   VAR 
      statConfiguration : "typeLPMLV30_Configuration" := ([12(false), 20(true)], [32(0)]);   // FB configuration
      statUnitModeChangeRequest : Bool := false;   // TRUE: Enable change into requested unit mode
      statCmdChangeRequest : Bool := false;   // TRUE: Enable change into requested state
      statFirstCycle { ExternalAccessible := 'False'; ExternalVisible := 'False'; ExternalWritable := 'False'} : Bool := true;   // First cycle of run
      statSCOld { ExternalAccessible := 'False'; ExternalVisible := 'False'; ExternalWritable := 'False'} : Bool := false;   // For edge detection
      statUnitMode { ExternalAccessible := 'False'; ExternalVisible := 'False'; ExternalWritable := 'False'} : DInt := "LPMLV30_MODE_MANUAL";   // Current command mode
      statUnitModeOld { ExternalAccessible := 'False'; ExternalVisible := 'False'; ExternalWritable := 'False'} : DInt := "LPMLV30_MODE_MANUAL";   // For edge detection
      statUnitModeCurrentInternal { ExternalAccessible := 'False'; ExternalVisible := 'False'; ExternalWritable := 'False'} : DInt := "LPMLV30_MODE_MANUAL";   // Current internal Mode
      statUnitModeCurrentInternalOld { ExternalAccessible := 'False'; ExternalVisible := 'False'; ExternalWritable := 'False'} : DInt := "LPMLV30_MODE_INVALID";   // For edge detection
      statStateCurrentOld { ExternalAccessible := 'False'; ExternalVisible := 'False'; ExternalWritable := 'False'} : DInt := "LPMLV30_STATE_STOPPED";   // For edge detection
      statStateInternal { ExternalAccessible := 'False'; ExternalVisible := 'False'; ExternalWritable := 'False'} : DInt := "LPMLV30_STATE_STOPPED";   // Current internal state
      statStateInternalOld { ExternalAccessible := 'False'; ExternalVisible := 'False'; ExternalWritable := 'False'} : DInt := "LPMLV30_STATE_UNDEFINED";   // For edge detection
      statCntrlCmdOld { ExternalAccessible := 'False'; ExternalVisible := 'False'; ExternalWritable := 'False'} : DInt := "LPMLV30_CMD_UNDEFINED";   // For edge detection
      statStatesInCurrentMode : Struct   // Copied from configuration
         clearing : Bool;
         stopped : Bool;
         starting : Bool;
         idle : Bool;
         suspended : Bool;
         execute : Bool;
         stopping : Bool;
         aborting : Bool;
         aborted : Bool;
         holding : Bool;
         held : Bool;
         unholding : Bool;
         suspending : Bool;
         unsuspending : Bool;
         resetting : Bool;
         completing : Bool;
         complete : Bool;
      END_STRUCT;
      statBooleanInterfaceModeOld { ExternalAccessible := 'False'; ExternalVisible := 'False'; ExternalWritable := 'False'} : DWord;   // For edge detection
      statBooleanInterfaceCmdOld { ExternalAccessible := 'False'; ExternalVisible := 'False'; ExternalWritable := 'False'} : Word;   // For edge detection
      statCmdChangeRequestOld : Bool := false;   // For edge detection
      statUnitModeChangeRequestOld : Bool := false;   // For edge detection
   END_VAR

   VAR_TEMP 
      tempCntrlCmd : DInt;   // Temporary control command
      tempBooleanInterfaceMode : DWord;   // Status of boolean Mode inputs if  boolean interface is active
      tempBooleanInterfaceCmd : Word;   // Status of boolean Cmd inputs except abort and stop if  boolean interface is active
      tempSCInternal : Bool;   // Internal state complete
      tempRetVal : Int;   // Tag for system function
      tempDiagnosticsBufferIndex : Int;   // Index of actual diagnostics buffer entry
      tempDiagnosticsBufferIndexSC : Int;   // Index of actual diagnostics buffer entry for SC messages
      tempDiagnosticsBufferIndexCmd : Int;   // Index of actual diagnostics buffer entry for control command messages
   END_VAR

   VAR CONSTANT 
      MSG_NO_MESSAGE : Byte := 16#00;   // Initial value
      MSG_MODE_CHANGED_SUCCESSFULLY : Byte := 16#01;   // Unit mode changed successfully
      MSG_STATE_CHANGED_SUCCESSFULLY : Byte := 16#02;   // State changed successfully
      MSG_MODE_ALREADY_ACTIVE : Byte := 16#03;   // Requested unit mode already active
      MSG_MODE_NOT_DEFINED : Byte := 16#80;   // Unit mode not defined
      MSG_CMD_NOT_DEFINED : Byte := 16#81;   // Control command not defined
      MSG_REQ_MODE_NOT_CONFIGURED : Byte := 16#82;   // Requested unit mode not configured
      MSG_MODE_TRANSITION_NOT_ALLOWED : Byte := 16#83;   // Unit mode transition not allowed
      MSG_CMD_NOT_ALLOWED : Byte := 16#84;   // Control command in this state not allowed
      MSG_SC_NOT_ALLOWED : Byte := 16#85;   // SC in this state not allowed
      MSG_STATE_CONFIG_FORCED : Byte := 16#86;   // State configuration forced to OMAC standard (corrected configuration -> FB output StatesDisabled)
   END_VAR


BEGIN
	//============================================================================================================
	// SIEMENS AG
	// (c)Copyright 2015 All Rights Reserved
	//------------------------------------------------------------------------------------------------------------
	// Library: LPMLV30
	// Tested with: S7-1200 with FW version V4.1, S7-1500 with FW version V1.7
	// Engineering: TIA Portal V13 SP1
	// Restrictions: ---
	// Requirements: S7-1200 / S7-1500
	// Functionality: Management of unit modes and states according to ISA TR88.00.02 - June 4, 2014
	//------------------------------------------------------------------------------------------------------------
	// Change log table:
	// Version  Date        Expert in charge    Changes applied
	// 03.00.01 29.05.2015  RK                  First released version 
	//============================================================================================================
	// Function block: LPMLV30_UnitModeStateManager
	//============================================================================================================
	
	IF NOT #statCmdChangeRequest AND #statCmdChangeRequestOld THEN // Falling edge CmdChangeRequest
	  #statCntrlCmdOld := "LPMLV30_CMD_UNDEFINED";
	END_IF;
	#statCmdChangeRequestOld := #statCmdChangeRequest;
	
	IF NOT #statUnitModeChangeRequest AND #statUnitModeChangeRequestOld THEN // Falling edge UnitModeChangeRequest
	  #statUnitModeOld := "LPMLV30_MODE_INVALID";
	END_IF;
	#statUnitModeChangeRequestOld := #statUnitModeChangeRequest;
	
	#tempDiagnosticsBufferIndex    := #diagnostics.bufferIndex; // Work with temporary variable during block execution
	#tempDiagnosticsBufferIndexSC  := -1;
	#tempDiagnosticsBufferIndexCmd := -1;
	
	IF #statFirstCycle THEN // Initialize values in first cycle
	  #tempDiagnosticsBufferIndex := -1;
	
	  #statConfiguration := #configuration; // Copy configuration from input
	  #statConfiguration.disabledUnitModes["LPMLV30_MODE_MANUAL"] := FALSE; // Unit mode Manual is mandatory
	  
	  // Initialize unit mode
	  #statUnitMode                   := "LPMLV30_MODE_MANUAL";
	  #statUnitModeOld                := "LPMLV30_MODE_MANUAL";
	  #UnitModeCurrent                := "LPMLV30_MODE_MANUAL";
	  #statUnitModeCurrentInternal    := "LPMLV30_MODE_MANUAL";
	  #statUnitModeCurrentInternalOld := "LPMLV30_MODE_INVALID";
	  #statBooleanInterfaceModeOld    := 0;
	  
	  // Initialize state
	  #StateCurrent         := "LPMLV30_STATE_STOPPED";
	  #StateRequested       := "LPMLV30_STATE_STOPPED";
	  #statStateInternal    := "LPMLV30_STATE_STOPPED";
	  #statStateInternalOld := "LPMLV30_STATE_UNDEFINED";
	  #statStateCurrentOld  := "LPMLV30_STATE_STOPPED";
	  
	  // Initialize control command
	  #tempCntrlCmd               := "LPMLV30_CMD_UNDEFINED";
	  #statCntrlCmdOld            := "LPMLV30_CMD_UNDEFINED";
	  #statBooleanInterfaceCmdOld := 0;
	END_IF; // End: Initialize values in first cycle
	
	//--------------------------------------------------------------------------------------------------
	// Evaluation of input parameters -> UnitMode, CntrlCmd
	//--------------------------------------------------------------------------------------------------
	IF NOT #statFirstCycle THEN // As from second cycle
	  IF NOT #enableBooleanInterface THEN // Set unit mode and control command according to input parameters
	    #statUnitMode := #UnitMode;
	    #tempCntrlCmd := #CntrlCmd;
	    
	    // Set change requests from input
	    #statUnitModeChangeRequest := #UnitModeChangeRequest;
	    #statCmdChangeRequest      := #CmdChangeRequest;
	  ELSE // Read boolean interface inputs
	    #statUnitModeChangeRequest := TRUE; // Change request static TRUE
	    #statUnitMode              := "LPMLV30_MODE_INVALID";
	    #tempBooleanInterfaceMode  := 0;
	    
	    // Collect unit mode from boolean inputs
	    #tempBooleanInterfaceMode.%X1  := #ProductionModeRequest;
	    #tempBooleanInterfaceMode.%X2  := #MaintenanceModeRequest;
	    #tempBooleanInterfaceMode.%X3  := #ManualModeRequest;
	    #tempBooleanInterfaceMode.%X4  := #UserMode01Request;
	    #tempBooleanInterfaceMode.%X5  := #UserMode02Request;
	    #tempBooleanInterfaceMode.%X6  := #UserMode03Request;
	    #tempBooleanInterfaceMode.%X7  := #UserMode04Request;
	    #tempBooleanInterfaceMode.%X8  := #UserMode05Request;
	    #tempBooleanInterfaceMode.%X9  := #UserMode06Request;
	    #tempBooleanInterfaceMode.%X10 := #UserMode07Request;
	    #tempBooleanInterfaceMode.%X11 := #UserMode08Request;
	    // #tempBooleanInterfaceMode.%X12 := #UserMode09Request;
	    // #tempBooleanInterfaceMode.%X13 := #UserMode10Request;
	    // #tempBooleanInterfaceMode.%X14 := #UserMode11Request;
	    // #tempBooleanInterfaceMode.%X15 := #UserMode12Request;
	    // #tempBooleanInterfaceMode.%X16 := #UserMode13Request;
	    // #tempBooleanInterfaceMode.%X17 := #UserMode14Request;
	    // #tempBooleanInterfaceMode.%X18 := #UserMode15Request;
	    // #tempBooleanInterfaceMode.%X19 := #UserMode16Request;
	    // #tempBooleanInterfaceMode.%X20 := #UserMode17Request;
	    // #tempBooleanInterfaceMode.%X21 := #UserMode18Request;
	    // #tempBooleanInterfaceMode.%X22 := #UserMode19Request;
	    // #tempBooleanInterfaceMode.%X23 := #UserMode20Request;
	    // #tempBooleanInterfaceMode.%X24 := #UserMode21Request;
	    // #tempBooleanInterfaceMode.%X25 := #UserMode22Request;
	    // #tempBooleanInterfaceMode.%X26 := #UserMode23Request;
	    // #tempBooleanInterfaceMode.%X27 := #UserMode24Request;
	    // #tempBooleanInterfaceMode.%X28 := #UserMode25Request;
	    // #tempBooleanInterfaceMode.%X29 := #UserMode26Request;
	    // #tempBooleanInterfaceMode.%X30 := #UserMode27Request;
	    // #tempBooleanInterfaceMode.%X31 := #UserMode28Request;
	
	    // Selection indicator: Rising edge at input, Priority (in case of multiple selection): Manual, Maintenance, User Mode 01..28, Production
	    IF #tempBooleanInterfaceMode.%X3  AND NOT #statBooleanInterfaceModeOld.%X3  THEN
	      #statUnitMode := "LPMLV30_MODE_MANUAL";
	    ELSIF #tempBooleanInterfaceMode.%X2  AND NOT #statBooleanInterfaceModeOld.%X2  THEN
	      #statUnitMode := "LPMLV30_MODE_MAINTENANCE";
	    ELSIF #tempBooleanInterfaceMode.%X4  AND NOT #statBooleanInterfaceModeOld.%X4  THEN
	      #statUnitMode := "LPMLV30_MODE_USER_01";
	    ELSIF #tempBooleanInterfaceMode.%X5  AND NOT #statBooleanInterfaceModeOld.%X5  THEN
	      #statUnitMode := "LPMLV30_MODE_USER_02";
	    ELSIF #tempBooleanInterfaceMode.%X6  AND NOT #statBooleanInterfaceModeOld.%X6  THEN
	      #statUnitMode := "LPMLV30_MODE_USER_03";
	    ELSIF #tempBooleanInterfaceMode.%X7  AND NOT #statBooleanInterfaceModeOld.%X7  THEN
	      #statUnitMode := "LPMLV30_MODE_USER_04";
	    ELSIF #tempBooleanInterfaceMode.%X8  AND NOT #statBooleanInterfaceModeOld.%X8  THEN
	      #statUnitMode := "LPMLV30_MODE_USER_05";
	    ELSIF #tempBooleanInterfaceMode.%X9  AND NOT #statBooleanInterfaceModeOld.%X9  THEN
	      #statUnitMode := "LPMLV30_MODE_USER_06";
	    ELSIF #tempBooleanInterfaceMode.%X10 AND NOT #statBooleanInterfaceModeOld.%X10 THEN
	      #statUnitMode := "LPMLV30_MODE_USER_07";
	    ELSIF #tempBooleanInterfaceMode.%X11 AND NOT #statBooleanInterfaceModeOld.%X11 THEN
	      #statUnitMode := "LPMLV30_MODE_USER_08";
	    ELSIF #tempBooleanInterfaceMode.%X12 AND NOT #statBooleanInterfaceModeOld.%X12 THEN
	      #statUnitMode := "LPMLV30_MODE_USER_09";
	    ELSIF #tempBooleanInterfaceMode.%X13 AND NOT #statBooleanInterfaceModeOld.%X13 THEN
	      #statUnitMode := "LPMLV30_MODE_USER_10";
	    ELSIF #tempBooleanInterfaceMode.%X14 AND NOT #statBooleanInterfaceModeOld.%X14 THEN
	      #statUnitMode := "LPMLV30_MODE_USER_11";
	    ELSIF #tempBooleanInterfaceMode.%X15 AND NOT #statBooleanInterfaceModeOld.%X15 THEN
	      #statUnitMode := "LPMLV30_MODE_USER_12";
	    ELSIF #tempBooleanInterfaceMode.%X16 AND NOT #statBooleanInterfaceModeOld.%X16 THEN
	      #statUnitMode := "LPMLV30_MODE_USER_13";
	    ELSIF #tempBooleanInterfaceMode.%X17 AND NOT #statBooleanInterfaceModeOld.%X17 THEN
	      #statUnitMode := "LPMLV30_MODE_USER_14";
	    ELSIF #tempBooleanInterfaceMode.%X18 AND NOT #statBooleanInterfaceModeOld.%X18 THEN
	      #statUnitMode := "LPMLV30_MODE_USER_15";
	    ELSIF #tempBooleanInterfaceMode.%X19 AND NOT #statBooleanInterfaceModeOld.%X19 THEN
	      #statUnitMode := "LPMLV30_MODE_USER_16";
	    ELSIF #tempBooleanInterfaceMode.%X20 AND NOT #statBooleanInterfaceModeOld.%X20 THEN
	      #statUnitMode := "LPMLV30_MODE_USER_17";
	    ELSIF #tempBooleanInterfaceMode.%X21 AND NOT #statBooleanInterfaceModeOld.%X21 THEN
	      #statUnitMode := "LPMLV30_MODE_USER_18";
	    ELSIF #tempBooleanInterfaceMode.%X22 AND NOT #statBooleanInterfaceModeOld.%X22 THEN
	      #statUnitMode := "LPMLV30_MODE_USER_19";
	    ELSIF #tempBooleanInterfaceMode.%X23 AND NOT #statBooleanInterfaceModeOld.%X23 THEN
	      #statUnitMode := "LPMLV30_MODE_USER_20";
	    ELSIF #tempBooleanInterfaceMode.%X24 AND NOT #statBooleanInterfaceModeOld.%X24 THEN
	      #statUnitMode := "LPMLV30_MODE_USER_21";
	    ELSIF #tempBooleanInterfaceMode.%X25 AND NOT #statBooleanInterfaceModeOld.%X25 THEN
	      #statUnitMode := "LPMLV30_MODE_USER_22";
	    ELSIF #tempBooleanInterfaceMode.%X26 AND NOT #statBooleanInterfaceModeOld.%X26 THEN
	      #statUnitMode := "LPMLV30_MODE_USER_23";
	    ELSIF #tempBooleanInterfaceMode.%X27 AND NOT #statBooleanInterfaceModeOld.%X27 THEN
	      #statUnitMode := "LPMLV30_MODE_USER_24";
	    ELSIF #tempBooleanInterfaceMode.%X28 AND NOT #statBooleanInterfaceModeOld.%X28 THEN
	      #statUnitMode := "LPMLV30_MODE_USER_25";
	    ELSIF #tempBooleanInterfaceMode.%X29 AND NOT #statBooleanInterfaceModeOld.%X29 THEN
	      #statUnitMode := "LPMLV30_MODE_USER_26";
	    ELSIF #tempBooleanInterfaceMode.%X30 AND NOT #statBooleanInterfaceModeOld.%X30 THEN
	      #statUnitMode := "LPMLV30_MODE_USER_27";
	    ELSIF #tempBooleanInterfaceMode.%X31 AND NOT #statBooleanInterfaceModeOld.%X31 THEN
	      #statUnitMode := "LPMLV30_MODE_USER_28";
	    ELSIF    #tempBooleanInterfaceMode.%X1  AND NOT #statBooleanInterfaceModeOld.%X1  THEN
	      #statUnitMode := "LPMLV30_MODE_PRODUCTION";
	    END_IF;
	    #statBooleanInterfaceModeOld := #tempBooleanInterfaceMode; // Save values for edge detection
	
	    // Evaluate CntrlCmd in boolean interface; priority descending: abort, stop, other commands
	    #statCmdChangeRequest    := TRUE; // Change request static TRUE
	    #tempBooleanInterfaceCmd := 0;
	
	    #tempBooleanInterfaceCmd.%X1  := #ResetCmdRequest;
	    #tempBooleanInterfaceCmd.%X2  := #StartCmdRequest;
	    #tempBooleanInterfaceCmd.%X4  := #HoldCmdRequest;
	    #tempBooleanInterfaceCmd.%X5  := #UnholdCmdRequest;
	    #tempBooleanInterfaceCmd.%X6  := #SuspendCmdRequest;
	    #tempBooleanInterfaceCmd.%X7  := #UnsuspendCmdRequest;
	    #tempBooleanInterfaceCmd.%X9  := #ClearCmdRequest;
	    #tempBooleanInterfaceCmd.%X10 := #CompleteCmdRequest; // Remember, complete command is not specified in the OMAC standard
	    
	    IF #AbortCmdRequest THEN
	      #tempCntrlCmd := "LPMLV30_CMD_ABORT";
	    ELSIF #StopCmdRequest THEN
	      #tempCntrlCmd := "LPMLV30_CMD_STOP";
	    ELSE
	      #tempCntrlCmd := "LPMLV30_CMD_UNDEFINED";
	
	      // Selection indicator: Rising edge at input, Priority (in case of multiple selection): complete, reset, start, hold, unhold, suspend, unsuspend, clear
	      IF    #tempBooleanInterfaceCmd.%X10 AND NOT #statBooleanInterfaceCmdOld.%X10 THEN
	        #tempCntrlCmd := "LPMLV30_CMD_COMPLETE";
	      ELSIF #tempBooleanInterfaceCmd.%X1  AND NOT #statBooleanInterfaceCmdOld.%X1  THEN
	        #tempCntrlCmd := "LPMLV30_CMD_RESET";
	      ELSIF #tempBooleanInterfaceCmd.%X2  AND NOT #statBooleanInterfaceCmdOld.%X2  THEN
	        #tempCntrlCmd := "LPMLV30_CMD_START";
	      ELSIF #tempBooleanInterfaceCmd.%X4  AND NOT #statBooleanInterfaceCmdOld.%X4  THEN
	        #tempCntrlCmd := "LPMLV30_CMD_HOLD";
	      ELSIF #tempBooleanInterfaceCmd.%X5  AND NOT #statBooleanInterfaceCmdOld.%X5  THEN
	        #tempCntrlCmd := "LPMLV30_CMD_UNHOLD";
	      ELSIF #tempBooleanInterfaceCmd.%X6  AND NOT #statBooleanInterfaceCmdOld.%X6  THEN
	        #tempCntrlCmd := "LPMLV30_CMD_SUSPEND";
	      ELSIF #tempBooleanInterfaceCmd.%X7  AND NOT #statBooleanInterfaceCmdOld.%X7  THEN
	        #tempCntrlCmd := "LPMLV30_CMD_UNSUSPEND";
	      ELSIF #tempBooleanInterfaceCmd.%X9  AND NOT #statBooleanInterfaceCmdOld.%X9  THEN
	        #tempCntrlCmd := "LPMLV30_CMD_CLEAR";
	      END_IF;
	    END_IF; // End: abort or stop cmd
	
	    #statBooleanInterfaceCmdOld := #tempBooleanInterfaceCmd; // Save values for edge detection
	  END_IF; // End: boolean interface
	END_IF; // End: As from second cycle
	// End: Evaluation of input parameters -> UnitMode, CntrlCmd
	
	//--------------------------------------------------------------------------------------------------
	// Unit mode manager
	//--------------------------------------------------------------------------------------------------
	IF NOT #statFirstCycle THEN // As from second cycle
	  //------------------------------------------------
	  //Message handling for mode manager: head part
	  //------------------------------------------------
	  IF #statUnitModeChangeRequest AND #statUnitMode <> #statUnitModeOld AND #statUnitMode <> "LPMLV30_MODE_INVALID" THEN
	    #tempDiagnosticsBufferIndex := #tempDiagnosticsBufferIndex + 1; // Next buffer index
	    IF #tempDiagnosticsBufferIndex > "LPMLV30_DIAG_BUFFER_UPPER_LIM" THEN
	      #tempDiagnosticsBufferIndex := 0;
	    END_IF;
	    // Check for defined unit modes
	    #tempRetVal := RD_SYS_T(#diagnostics.buffer[#tempDiagnosticsBufferIndex].timestamp);
	    #diagnostics.buffer[#tempDiagnosticsBufferIndex].UnitModeCurrent := DINT_TO_BYTE(#UnitModeCurrent);
	    #diagnostics.buffer[#tempDiagnosticsBufferIndex].StateCurrent    := DINT_TO_BYTE(#StateCurrent);
	    #diagnostics.buffer[#tempDiagnosticsBufferIndex].UnitMode := DINT_TO_BYTE(#statUnitMode);
	    #diagnostics.buffer[#tempDiagnosticsBufferIndex].CntrlCmd := DINT_TO_BYTE(#tempCntrlCmd);
	    #diagnostics.buffer[#tempDiagnosticsBufferIndex].SC := #SC;
	    #diagnostics.buffer[#tempDiagnosticsBufferIndex].message := #MSG_NO_MESSAGE;
	    
	    IF #statUnitMode < "LPMLV30_MODE_INVALID" OR #statUnitMode > "LPMLV30_MODE_USER_28" THEN
	      #diagnostics.buffer[#tempDiagnosticsBufferIndex].message := #MSG_MODE_NOT_DEFINED;
	    ELSIF #statUnitMode = #statUnitModeCurrentInternal THEN
	      #diagnostics.buffer[#tempDiagnosticsBufferIndex].message := #MSG_MODE_ALREADY_ACTIVE;
	    END_IF;
	  END_IF; // End: message handling for mode manager: head part
	END_IF; // End: As from second cycle
	
	//------------------------------------------------
	// Unit mode machine
	//------------------------------------------------
	// Check if unit mode has to be changed
	IF (#statUnitModeChangeRequest AND
	  #statUnitMode <> #statUnitModeCurrentInternal AND
	  #statUnitMode <> #statUnitModeOld AND
	  #statUnitMode > "LPMLV30_MODE_INVALID" AND
	  #statUnitMode <= "LPMLV30_MODE_USER_28"
	  ) OR
	  #statFirstCycle
	THEN
	  // Check if state is available
	  IF #statStateInternal = "LPMLV30_STATE_EXECUTE" OR //  Every state but not in execute
	    #statStateInternal <> #StateRequested // Means to be in wait state or target state             
	  THEN
	    #diagnostics.buffer[#tempDiagnosticsBufferIndex].message := #MSG_MODE_TRANSITION_NOT_ALLOWED;
	  ELSE
	    IF #statConfiguration.disabledUnitModes[#statUnitMode] = FALSE THEN
	      // State in target unit mode available
	      IF ((NOT #statConfiguration.disabledStatesInUnitModes[#statUnitMode].%X17 = FALSE) AND (#statStateInternal = "LPMLV30_STATE_COMPLETE")) OR
	        ((NOT #statConfiguration.disabledStatesInUnitModes[#statUnitMode].%X11 = FALSE) AND (#statStateInternal = "LPMLV30_STATE_HELD")) OR
	        ((NOT #statConfiguration.disabledStatesInUnitModes[#statUnitMode].%X5 = FALSE) AND (#statStateInternal = "LPMLV30_STATE_SUSPENDED"))
	      THEN
	        #diagnostics.buffer[#tempDiagnosticsBufferIndex].message := #MSG_MODE_TRANSITION_NOT_ALLOWED;
	      ELSE
	        // Set outputs
	        #UnitModeChangeInProcess := TRUE;
	        #UnitModeRequested := #statUnitMode;
	        // Set internal variable
	        #statUnitModeCurrentInternal := #statUnitMode;
	
	        // Read current configuration for state
	        #statStatesInCurrentMode.clearing := NOT #statConfiguration.disabledStatesInUnitModes[#statUnitMode].%X1;
	        #statStatesInCurrentMode.stopped := NOT #statConfiguration.disabledStatesInUnitModes[#statUnitMode].%X2;
	        #statStatesInCurrentMode.starting := NOT #statConfiguration.disabledStatesInUnitModes[#statUnitMode].%X3;
	        #statStatesInCurrentMode.idle := NOT #statConfiguration.disabledStatesInUnitModes[#statUnitMode].%X4;
	        #statStatesInCurrentMode.suspended := NOT #statConfiguration.disabledStatesInUnitModes[#statUnitMode].%X5;
	        #statStatesInCurrentMode.execute := NOT #statConfiguration.disabledStatesInUnitModes[#statUnitMode].%X6;
	        #statStatesInCurrentMode.stopping := NOT #statConfiguration.disabledStatesInUnitModes[#statUnitMode].%X7;
	        #statStatesInCurrentMode.aborting := NOT #statConfiguration.disabledStatesInUnitModes[#statUnitMode].%X8;
	        #statStatesInCurrentMode.aborted := NOT #statConfiguration.disabledStatesInUnitModes[#statUnitMode].%X9;
	        #statStatesInCurrentMode.holding := NOT #statConfiguration.disabledStatesInUnitModes[#statUnitMode].%X10;
	        #statStatesInCurrentMode.held := NOT #statConfiguration.disabledStatesInUnitModes[#statUnitMode].%X11;
	        #statStatesInCurrentMode.unholding := NOT #statConfiguration.disabledStatesInUnitModes[#statUnitMode].%X12;
	        #statStatesInCurrentMode.suspending := NOT #statConfiguration.disabledStatesInUnitModes[#statUnitMode].%X13;
	        #statStatesInCurrentMode.unsuspending := NOT #statConfiguration.disabledStatesInUnitModes[#statUnitMode].%X14;
	        #statStatesInCurrentMode.resetting := NOT #statConfiguration.disabledStatesInUnitModes[#statUnitMode].%X15;
	        #statStatesInCurrentMode.completing := NOT #statConfiguration.disabledStatesInUnitModes[#statUnitMode].%X16;
	        #statStatesInCurrentMode.complete := NOT #statConfiguration.disabledStatesInUnitModes[#statUnitMode].%X17;
	      END_IF; // End: state in target unit mode available
	    ELSE
	      #diagnostics.buffer[#tempDiagnosticsBufferIndex].message := #MSG_REQ_MODE_NOT_CONFIGURED;
	    END_IF;
	  END_IF;
	
	  // Set the minimum required states for every unit mode
	  IF NOT #statStatesInCurrentMode.stopped OR
	    NOT #statStatesInCurrentMode.idle OR
	    NOT #statStatesInCurrentMode.execute OR
	    NOT #statStatesInCurrentMode.aborted OR
	    NOT #statStatesInCurrentMode.resetting OR
	    NOT #statStatesInCurrentMode.starting OR
	    NOT #statStatesInCurrentMode.stopping OR
	    NOT #statStatesInCurrentMode.clearing OR
	    NOT #statStatesInCurrentMode.aborting OR
	    (NOT #statStatesInCurrentMode.complete AND #statStatesInCurrentMode.completing) OR
	    (NOT #statStatesInCurrentMode.suspended AND (#statStatesInCurrentMode.suspending OR #statStatesInCurrentMode.unsuspending)) OR
	    (NOT #statStatesInCurrentMode.held AND (#statStatesInCurrentMode.holding OR #statStatesInCurrentMode.unholding))
	  THEN
	    #statStatesInCurrentMode.stopped := TRUE;
	    #statStatesInCurrentMode.idle := TRUE;
	    #statStatesInCurrentMode.execute := TRUE;
	    #statStatesInCurrentMode.aborted := TRUE;
	    
	    #statStatesInCurrentMode.resetting := TRUE;
	    #statStatesInCurrentMode.starting := TRUE;
	    #statStatesInCurrentMode.aborting := TRUE;
	    #statStatesInCurrentMode.stopping := TRUE;
	    #statStatesInCurrentMode.clearing := TRUE;
	    
	    // Held
	    IF NOT #statStatesInCurrentMode.held
	      AND (#statStatesInCurrentMode.holding OR #statStatesInCurrentMode.unholding)
	    THEN
	      #statStatesInCurrentMode.held := TRUE;
	      #statStatesInCurrentMode.holding := TRUE;
	      #statStatesInCurrentMode.unholding := TRUE;
	    END_IF;
	    // Suspended
	    IF NOT #statStatesInCurrentMode.suspended
	      AND (#statStatesInCurrentMode.suspending OR #statStatesInCurrentMode.unsuspending)
	    THEN
	      #statStatesInCurrentMode.suspended := TRUE;
	      #statStatesInCurrentMode.suspending := TRUE;
	      #statStatesInCurrentMode.unsuspending := TRUE;
	    END_IF;
	    // Complete
	    IF NOT #statStatesInCurrentMode.complete
	      AND #statStatesInCurrentMode.completing
	    THEN
	      #statStatesInCurrentMode.complete := TRUE;
	      #statStatesInCurrentMode.completing := TRUE;
	    END_IF;
	    
	    #tempDiagnosticsBufferIndex := #tempDiagnosticsBufferIndex + 1; // Next buffer index
	    IF #tempDiagnosticsBufferIndex > "LPMLV30_DIAG_BUFFER_UPPER_LIM" THEN
	      #tempDiagnosticsBufferIndex := 0;
	    END_IF;
	    
	    // Write diagnostics
	    #tempRetVal := RD_SYS_T(#diagnostics.buffer[#tempDiagnosticsBufferIndex].timestamp);
	    #diagnostics.buffer[#tempDiagnosticsBufferIndex].UnitModeCurrent := DINT_TO_BYTE(#UnitModeCurrent);
	    #diagnostics.buffer[#tempDiagnosticsBufferIndex].StateCurrent    := DINT_TO_BYTE(#StateCurrent);
	    #diagnostics.buffer[#tempDiagnosticsBufferIndex].UnitMode := DINT_TO_BYTE(#statUnitMode);
	    #diagnostics.buffer[#tempDiagnosticsBufferIndex].CntrlCmd := DINT_TO_BYTE(#tempCntrlCmd);
	    #diagnostics.buffer[#tempDiagnosticsBufferIndex].SC := #SC;
	    #diagnostics.buffer[#tempDiagnosticsBufferIndex].message := #MSG_STATE_CONFIG_FORCED;
	  END_IF; // End: set the minimum required states for every unit mode
	  
	  #UnitModeCurrent := #statUnitModeCurrentInternal; // Write current unit mode on output
	  
	  // Write correct state configuration of current mode
	  #StatesDisabled.%X1 := NOT #statStatesInCurrentMode.clearing;
	  #StatesDisabled.%X2 := NOT #statStatesInCurrentMode.stopped;
	  #StatesDisabled.%X3 := NOT #statStatesInCurrentMode.starting;
	  #StatesDisabled.%X4 := NOT #statStatesInCurrentMode.idle;
	  #StatesDisabled.%X5 := NOT #statStatesInCurrentMode.suspended;
	  #StatesDisabled.%X6 := NOT #statStatesInCurrentMode.execute;
	  #StatesDisabled.%X7 := NOT #statStatesInCurrentMode.stopping;
	  #StatesDisabled.%X8 := NOT #statStatesInCurrentMode.aborting;
	  #StatesDisabled.%X9 := NOT #statStatesInCurrentMode.aborted;
	  #StatesDisabled.%X10 := NOT #statStatesInCurrentMode.holding;
	  #StatesDisabled.%X11 := NOT #statStatesInCurrentMode.held;
	  #StatesDisabled.%X12 := NOT #statStatesInCurrentMode.unholding;
	  #StatesDisabled.%X13 := NOT #statStatesInCurrentMode.suspending;
	  #StatesDisabled.%X14 := NOT #statStatesInCurrentMode.unsuspending;
	  #StatesDisabled.%X15 := NOT #statStatesInCurrentMode.resetting;
	  #StatesDisabled.%X16 := NOT #statStatesInCurrentMode.completing;
	  #StatesDisabled.%X17 := NOT #statStatesInCurrentMode.complete;
	  
	  //-----------------------------------------------
	  // Message handling for mode manager: foot part
	  //-----------------------------------------------
	  IF NOT #statFirstCycle THEN
	    IF #diagnostics.buffer[#tempDiagnosticsBufferIndex].message = #MSG_NO_MESSAGE THEN // ELSE: Unit mode wasn´t changed successfully
	      #diagnostics.buffer[#tempDiagnosticsBufferIndex].message := #MSG_MODE_CHANGED_SUCCESSFULLY;
	    END_IF;
	  END_IF;
	ELSE
	  #UnitModeChangeInProcess := FALSE; // No unit mode change
	END_IF;// End: check if unit mode has to be changed
	// End: Unit mode manager
	
	//--------------------------------------------------------------------------------------------------
	// State manager
	//--------------------------------------------------------------------------------------------------
	IF NOT #statFirstCycle THEN // As from second cycle
	  IF #SC AND NOT #statSCOld THEN // Detect a rising edge at state complete signal
	    #tempSCInternal := TRUE;
	  ELSE
	    #tempSCInternal := FALSE;
	  END_IF;
	  #statSCOld := #SC; // End: Detect a rising edge at state complete signal
	
	  //---------------------------------------------------------------------
	  // Message handling for state manager: head part 
	  //---------------------------------------------------------------------
	  IF #tempSCInternal THEN // Check if rising edge of SC was detected
	    #tempDiagnosticsBufferIndex := #tempDiagnosticsBufferIndex + 1; // Next buffer index
	    IF #tempDiagnosticsBufferIndex > "LPMLV30_DIAG_BUFFER_UPPER_LIM" THEN
	      #tempDiagnosticsBufferIndex := 0;
	    END_IF;
	    #tempDiagnosticsBufferIndexSC := #tempDiagnosticsBufferIndex;
	
	    // Check current state to use SC
	    IF #statStateInternal = "LPMLV30_STATE_CLEARING"    OR
	      #statStateInternal = "LPMLV30_STATE_STARTING"     OR
	      #statStateInternal = "LPMLV30_STATE_STOPPING"     OR
	      #statStateInternal = "LPMLV30_STATE_ABORTING"     OR
	      #statStateInternal = "LPMLV30_STATE_HOLDING"      OR
	      #statStateInternal = "LPMLV30_STATE_UNHOLDING"    OR
	      #statStateInternal = "LPMLV30_STATE_SUSPENDING"   OR
	      #statStateInternal = "LPMLV30_STATE_UNSUSPENDING" OR
	      #statStateInternal = "LPMLV30_STATE_RESETTING"    OR
	      #statStateInternal = "LPMLV30_STATE_COMPLETING"   OR
	      #statStateInternal = "LPMLV30_STATE_EXECUTE"
	    THEN // Write diagnostics     
	      #tempRetVal := RD_SYS_T(#diagnostics.buffer[#tempDiagnosticsBufferIndex].timestamp);
	      #diagnostics.buffer[#tempDiagnosticsBufferIndex].UnitModeCurrent := DINT_TO_BYTE(#UnitModeCurrent);
	      #diagnostics.buffer[#tempDiagnosticsBufferIndex].StateCurrent    := DINT_TO_BYTE(#StateCurrent);
	      #diagnostics.buffer[#tempDiagnosticsBufferIndex].UnitMode := DINT_TO_BYTE(#statUnitMode);
	      #diagnostics.buffer[#tempDiagnosticsBufferIndex].CntrlCmd := DINT_TO_BYTE(#tempCntrlCmd);
	      #diagnostics.buffer[#tempDiagnosticsBufferIndex].SC := #SC;
	      #diagnostics.buffer[#tempDiagnosticsBufferIndex].message := #MSG_NO_MESSAGE;
	    ELSE // Write diagnostics
	      #tempRetVal := RD_SYS_T(#diagnostics.buffer[#tempDiagnosticsBufferIndex].timestamp);
	      #diagnostics.buffer[#tempDiagnosticsBufferIndex].UnitModeCurrent := DINT_TO_BYTE(#UnitModeCurrent);
	      #diagnostics.buffer[#tempDiagnosticsBufferIndex].StateCurrent    := DINT_TO_BYTE(#StateCurrent);
	      #diagnostics.buffer[#tempDiagnosticsBufferIndex].UnitMode := DINT_TO_BYTE(#statUnitMode);
	      #diagnostics.buffer[#tempDiagnosticsBufferIndex].CntrlCmd := DINT_TO_BYTE(#tempCntrlCmd);
	      #diagnostics.buffer[#tempDiagnosticsBufferIndex].SC := #SC;
	      #diagnostics.buffer[#tempDiagnosticsBufferIndex].message := #MSG_SC_NOT_ALLOWED;
	    END_IF; // End: Check current state to use SC
	  END_IF;
	  
	  // Check if defined control command was sent correctly
	  IF #statCmdChangeRequest AND #tempCntrlCmd <> #statCntrlCmdOld AND #tempCntrlCmd <> "LPMLV30_CMD_UNDEFINED" THEN
	    IF #tempCntrlCmd = "LPMLV30_CMD_RESET"     OR
	       #tempCntrlCmd = "LPMLV30_CMD_START"     OR
	       #tempCntrlCmd = "LPMLV30_CMD_STOP"      OR
	       #tempCntrlCmd = "LPMLV30_CMD_HOLD"      OR
	       #tempCntrlCmd = "LPMLV30_CMD_UNHOLD"    OR
	       #tempCntrlCmd = "LPMLV30_CMD_SUSPEND"   OR
	       #tempCntrlCmd = "LPMLV30_CMD_UNSUSPEND" OR
	       #tempCntrlCmd = "LPMLV30_CMD_ABORT"     OR
	       #tempCntrlCmd = "LPMLV30_CMD_CLEAR"     OR
	       #tempCntrlCmd = "LPMLV30_CMD_COMPLETE" // Info: Complete command not in the OMAC standard
	    THEN
	      #tempDiagnosticsBufferIndex := #tempDiagnosticsBufferIndex + 1; // Next buffer index
	      IF #tempDiagnosticsBufferIndex > "LPMLV30_DIAG_BUFFER_UPPER_LIM" THEN
	        #tempDiagnosticsBufferIndex := 0;
	      END_IF;
	      #tempDiagnosticsBufferIndexCmd := #tempDiagnosticsBufferIndex;
	
	      // Write diagnostics
	      #tempRetVal := RD_SYS_T(#diagnostics.buffer[#tempDiagnosticsBufferIndex].timestamp);
	      #diagnostics.buffer[#tempDiagnosticsBufferIndex].UnitModeCurrent := DINT_TO_BYTE(#UnitModeCurrent);
	      #diagnostics.buffer[#tempDiagnosticsBufferIndex].StateCurrent    := DINT_TO_BYTE(#StateCurrent);
	      #diagnostics.buffer[#tempDiagnosticsBufferIndex].UnitMode := DINT_TO_BYTE(#statUnitMode);
	      #diagnostics.buffer[#tempDiagnosticsBufferIndex].CntrlCmd := DINT_TO_BYTE(#tempCntrlCmd);
	      #diagnostics.buffer[#tempDiagnosticsBufferIndex].SC := #SC;
	      #diagnostics.buffer[#tempDiagnosticsBufferIndex].message := #MSG_NO_MESSAGE;
	      // Write message if CntrlCmd is not allowed
	      IF ((#statStateInternal = "LPMLV30_STATE_CLEARING" OR
	        #statStateInternal = "LPMLV30_STATE_STARTING" OR
	        #statStateInternal = "LPMLV30_STATE_STOPPING" OR
	        #statStateInternal = "LPMLV30_STATE_ABORTING" OR
	        #statStateInternal = "LPMLV30_STATE_HOLDING" OR
	        #statStateInternal = "LPMLV30_STATE_UNHOLDING" OR
	        #statStateInternal = "LPMLV30_STATE_SUSPENDING" OR
	        #statStateInternal = "LPMLV30_STATE_UNSUSPENDING" OR
	        #statStateInternal = "LPMLV30_STATE_RESETTING" OR
	        #statStateInternal = "LPMLV30_STATE_COMPLETING") AND
	        NOT (#tempCntrlCmd = "LPMLV30_CMD_ABORT") AND NOT (#tempCntrlCmd = "LPMLV30_CMD_STOP")) OR
	        (#statStateInternal = "LPMLV30_STATE_ABORTED" AND (#tempCntrlCmd = "LPMLV30_CMD_ABORT"))
	      THEN
	        #diagnostics.buffer[#tempDiagnosticsBufferIndex].message := #MSG_CMD_NOT_ALLOWED;
	      END_IF;
	    ELSE
	      // Not defined control command was sent
	      #tempDiagnosticsBufferIndex := #tempDiagnosticsBufferIndex + 1; // Next buffer index
	      IF #tempDiagnosticsBufferIndex > "LPMLV30_DIAG_BUFFER_UPPER_LIM" THEN
	        #tempDiagnosticsBufferIndex := 0;
	      END_IF;
	      #tempDiagnosticsBufferIndexCmd := #tempDiagnosticsBufferIndex;
	
	      // Write diagnostics
	      #tempRetVal := RD_SYS_T(#diagnostics.buffer[#tempDiagnosticsBufferIndex].timestamp);
	      #diagnostics.buffer[#tempDiagnosticsBufferIndex].UnitModeCurrent := DINT_TO_BYTE(#UnitModeCurrent);
	      #diagnostics.buffer[#tempDiagnosticsBufferIndex].StateCurrent    := DINT_TO_BYTE(#StateCurrent);
	      #diagnostics.buffer[#tempDiagnosticsBufferIndex].UnitMode := DINT_TO_BYTE(#statUnitMode);
	      #diagnostics.buffer[#tempDiagnosticsBufferIndex].CntrlCmd := DINT_TO_BYTE(#tempCntrlCmd);
	      #diagnostics.buffer[#tempDiagnosticsBufferIndex].SC := #SC;
	      #diagnostics.buffer[#tempDiagnosticsBufferIndex].message := #MSG_CMD_NOT_DEFINED;
	    END_IF;
	  END_IF; // End: message handling for state manager: head part 
	  
	  //---------------------------------------------------------------------
	  // State machine
	  //---------------------------------------------------------------------
	  IF #statCmdChangeRequest AND #tempCntrlCmd <> #statCntrlCmdOld AND #tempCntrlCmd = "LPMLV30_CMD_ABORT" AND // Check if abort command was sent correctly    
	    #statStateInternal <> "LPMLV30_STATE_ABORTED" AND
	    #statStateInternal <> "LPMLV30_STATE_ABORTING"
	  THEN
	    // Abort command was sent correctly
	    #StateChangeInProcess := TRUE;
	    #StateRequested := "LPMLV30_STATE_ABORTED";
	    // Select next state
	    IF #statStatesInCurrentMode.aborting THEN
	      #statStateInternal := "LPMLV30_STATE_ABORTING";
	    ELSE
	      #statStateInternal := "LPMLV30_STATE_ABORTED";
	    END_IF;
	    
	  ELSIF #statCmdChangeRequest AND #tempCntrlCmd <> #statCntrlCmdOld AND #tempCntrlCmd = "LPMLV30_CMD_STOP" AND // Check if correct stop command was sent
	    #statStateInternal <> "LPMLV30_STATE_ABORTED"  AND
	    #statStateInternal <> "LPMLV30_STATE_ABORTING" AND
	    #statStateInternal <> "LPMLV30_STATE_CLEARING" AND
	    #statStateInternal <> "LPMLV30_STATE_STOPPING" AND
	    #statStateInternal <> "LPMLV30_STATE_STOPPED"
	  THEN
	    // Stop command was sent correctly
	    #StateChangeInProcess := TRUE;
	    #StateRequested := "LPMLV30_STATE_STOPPED";
	    // Select next state
	    IF #statStatesInCurrentMode.stopping THEN
	      #statStateInternal := "LPMLV30_STATE_STOPPING";
	    ELSE
	      #statStateInternal := "LPMLV30_STATE_STOPPED";
	    END_IF;
	    
	  ELSE // Internal state machine
	    CASE #statStateInternal OF
	      "LPMLV30_STATE_EXECUTE":
	        #StateChangeInProcess := FALSE;
	        // Check if state is completed
	        IF #tempSCInternal AND #statStatesInCurrentMode.completing THEN // ELSE: Wait for SC (state complete)
	          #StateChangeInProcess := TRUE;
	          #StateRequested    := "LPMLV30_STATE_COMPLETE";
	          #statStateInternal := "LPMLV30_STATE_COMPLETING";
	        ELSIF #tempSCInternal AND #statStatesInCurrentMode.complete THEN
	          #StateChangeInProcess := TRUE;
	          #StateRequested    := "LPMLV30_STATE_COMPLETE";
	          #statStateInternal := "LPMLV30_STATE_COMPLETE";
	        ELSIF #tempSCInternal AND NOT #statStatesInCurrentMode.completing AND NOT #statStatesInCurrentMode.complete THEN
	          #diagnostics.buffer[#tempDiagnosticsBufferIndexSC].message := #MSG_SC_NOT_ALLOWED;
	        END_IF;
	
	        IF #statCmdChangeRequest AND #tempCntrlCmd <> #statCntrlCmdOld AND #tempCntrlCmd <> "LPMLV30_CMD_UNDEFINED" AND
	          NOT (#tempSCInternal AND (#statStatesInCurrentMode.completing OR #statStatesInCurrentMode.complete))
	        THEN // Check if state change is requested
	          CASE #tempCntrlCmd OF // Check control command
	            "LPMLV30_CMD_COMPLETE": // Remember, the Complete command is not specified in the OMAC standard
	              // Check if valid state for command is in use by current unit mode
	              IF #statStatesInCurrentMode.completing THEN
	                #StateChangeInProcess := TRUE;
	                #StateRequested    := "LPMLV30_STATE_COMPLETE";
	                #statStateInternal := "LPMLV30_STATE_COMPLETING";
	              ELSIF #statStatesInCurrentMode.complete THEN
	                #StateChangeInProcess := TRUE;
	                #StateRequested    := "LPMLV30_STATE_COMPLETE";
	                #statStateInternal := "LPMLV30_STATE_COMPLETE";
	              ELSE
	                #diagnostics.buffer[#tempDiagnosticsBufferIndexCmd].message := #MSG_CMD_NOT_ALLOWED;
	              END_IF;
	              
	            "LPMLV30_CMD_RESET":
	              IF NOT #statStatesInCurrentMode.completing AND NOT #statStatesInCurrentMode.complete THEN
	                // Check if valid state for command is in use by current unit mode
	                IF #statStatesInCurrentMode.resetting THEN
	                  #StateChangeInProcess := TRUE;
	                  #StateRequested    := "LPMLV30_STATE_IDLE";
	                  #statStateInternal := "LPMLV30_STATE_RESETTING";
	                ELSIF #statStatesInCurrentMode.idle THEN
	                  #StateChangeInProcess := TRUE;
	                  #StateRequested    := "LPMLV30_STATE_IDLE";
	                  #statStateInternal := "LPMLV30_STATE_IDLE";
	                ELSE
	                  #diagnostics.buffer[#tempDiagnosticsBufferIndexCmd].message := #MSG_CMD_NOT_ALLOWED;
	                END_IF;
	              END_IF;
	              
	            "LPMLV30_CMD_HOLD":
	              // Check if valid state for command is in use by current unit mode
	              IF #statStatesInCurrentMode.holding THEN
	                #StateChangeInProcess := TRUE;
	                #StateRequested    := "LPMLV30_STATE_HELD";
	                #statStateInternal := "LPMLV30_STATE_HOLDING";
	              ELSIF #statStatesInCurrentMode.held THEN
	                #StateChangeInProcess := TRUE;
	                #StateRequested    := "LPMLV30_STATE_HELD";
	                #statStateInternal := "LPMLV30_STATE_HELD";
	              ELSE
	                #diagnostics.buffer[#tempDiagnosticsBufferIndexCmd].message := #MSG_CMD_NOT_ALLOWED;
	              END_IF;
	              
	            "LPMLV30_CMD_SUSPEND":
	              // Check if valid state for command is in use by current unit mode
	              IF #statStatesInCurrentMode.suspending THEN
	                #StateChangeInProcess := TRUE;
	                #StateRequested    := "LPMLV30_STATE_SUSPENDED";
	                #statStateInternal := "LPMLV30_STATE_SUSPENDING";
	              ELSIF #statStatesInCurrentMode.suspended THEN
	                #StateChangeInProcess := TRUE;
	                #StateRequested    := "LPMLV30_STATE_SUSPENDED";
	                #statStateInternal := "LPMLV30_STATE_SUSPENDED";
	              ELSE
	                #diagnostics.buffer[#tempDiagnosticsBufferIndexCmd].message := #MSG_CMD_NOT_ALLOWED;
	              END_IF;
	            ELSE
	              IF #diagnostics.buffer[#tempDiagnosticsBufferIndexCmd].message = #MSG_NO_MESSAGE THEN // ELSE: Message was already written in head part of message handling
	                #diagnostics.buffer[#tempDiagnosticsBufferIndexCmd].message := #MSG_CMD_NOT_ALLOWED;
	              END_IF;
	          END_CASE;
	        END_IF;
	        
	      "LPMLV30_STATE_COMPLETING":
	        // Check if state is completed
	        IF #tempSCInternal AND #statStatesInCurrentMode.complete THEN
	          #statStateInternal := "LPMLV30_STATE_COMPLETE";
	        ELSIF #tempSCInternal AND NOT #statStatesInCurrentMode.complete THEN
	          #diagnostics.buffer[#tempDiagnosticsBufferIndexSC].message := #MSG_SC_NOT_ALLOWED;
	        END_IF;
	        
	      "LPMLV30_STATE_COMPLETE":
	        #StateChangeInProcess := FALSE;
	        IF #statCmdChangeRequest AND #tempCntrlCmd <> #statCntrlCmdOld AND #tempCntrlCmd <> "LPMLV30_CMD_UNDEFINED" THEN // Check if state change is requested
	          CASE #tempCntrlCmd OF // Check control command
	            "LPMLV30_CMD_RESET":
	              // Check if valid state for command is in use by current unit mode
	              IF #statStatesInCurrentMode.resetting THEN
	                #StateChangeInProcess := TRUE;
	                #StateRequested    := "LPMLV30_STATE_IDLE";
	                #statStateInternal := "LPMLV30_STATE_RESETTING";
	              ELSIF #statStatesInCurrentMode.idle THEN
	                #StateChangeInProcess := TRUE;
	                #StateRequested    := "LPMLV30_STATE_IDLE";
	                #statStateInternal := "LPMLV30_STATE_IDLE";
	              ELSE
	                #diagnostics.buffer[#tempDiagnosticsBufferIndexCmd].message := #MSG_CMD_NOT_ALLOWED;
	              END_IF;
	              
	            "LPMLV30_CMD_START":
	              // Check if valid state for command is in use by current unit mode
	              IF NOT #statStatesInCurrentMode.resetting AND NOT #statStatesInCurrentMode.idle THEN
	                #StateChangeInProcess := TRUE;
	                #StateRequested := "LPMLV30_STATE_EXECUTE";
	                // Check if valid state for command is in use by current unit mode
	                IF #statStatesInCurrentMode.starting THEN
	                  #statStateInternal := "LPMLV30_STATE_STARTING";
	                ELSE
	                  #statStateInternal := "LPMLV30_STATE_EXECUTE";
	                END_IF;
	              ELSE
	                #diagnostics.buffer[#tempDiagnosticsBufferIndexCmd].message := #MSG_CMD_NOT_ALLOWED;
	              END_IF;
	            ELSE
	              IF #diagnostics.buffer[#tempDiagnosticsBufferIndexCmd].message = #MSG_NO_MESSAGE THEN // ELSE: Message was already written in head part of message handling
	                #diagnostics.buffer[#tempDiagnosticsBufferIndexCmd].message := #MSG_CMD_NOT_ALLOWED;
	              END_IF;
	          END_CASE;
	        END_IF;
	        
	      "LPMLV30_STATE_RESETTING":
	        // Check if state is completed
	        // No message handling needed -> Idle is minimum required state
	        IF #tempSCInternal THEN // ELSE: Wait for state complete signal
	          #statStateInternal := "LPMLV30_STATE_IDLE";
	        END_IF;
	        
	      "LPMLV30_STATE_IDLE":
	        #StateChangeInProcess := FALSE;
	        //  No message handling needed -> Execute is minimum required state
	        //  Check if valid command is sent
	        IF #statCmdChangeRequest AND #tempCntrlCmd <> #statCntrlCmdOld AND #tempCntrlCmd <> "LPMLV30_CMD_UNDEFINED" THEN // Check if state change is requested      
	          CASE #tempCntrlCmd OF // Check control command
	            "LPMLV30_CMD_START":
	              #StateChangeInProcess := TRUE;
	              #StateRequested := "LPMLV30_STATE_EXECUTE";
	              // Check if valid state for command is in use by current mode
	              IF #statStatesInCurrentMode.starting THEN
	                #statStateInternal := "LPMLV30_STATE_STARTING";
	              ELSE
	                #statStateInternal := "LPMLV30_STATE_EXECUTE";
	              END_IF;
	            ELSE
	              IF #diagnostics.buffer[#tempDiagnosticsBufferIndexCmd].message = #MSG_NO_MESSAGE THEN // ELSE: Message was already written in head part of message handling
	                #diagnostics.buffer[#tempDiagnosticsBufferIndexCmd].message := #MSG_CMD_NOT_ALLOWED;
	              END_IF;
	          END_CASE;
	        END_IF;
	        
	      "LPMLV30_STATE_STARTING",
	      "LPMLV30_STATE_UNHOLDING",
	      "LPMLV30_STATE_UNSUSPENDING":
	        // Check if state is completed
	        IF #tempSCInternal THEN // ELSE: Wait for state complete signal
	          #statStateInternal := "LPMLV30_STATE_EXECUTE";
	        END_IF;
	        
	      "LPMLV30_STATE_HOLDING":
	        // Check if state is completed
	        IF #tempSCInternal AND #statStatesInCurrentMode.held THEN // ELSE: Wait for state complete signal
	          #statStateInternal := "LPMLV30_STATE_HELD";
	        ELSIF #tempSCInternal AND NOT #statStatesInCurrentMode.held THEN
	          #diagnostics.buffer[#tempDiagnosticsBufferIndexSC].message := #MSG_SC_NOT_ALLOWED;
	        END_IF;
	        
	      "LPMLV30_STATE_HELD":
	        #StateChangeInProcess := FALSE;
	        //  Check if valid command is sent
	        IF #statCmdChangeRequest AND #tempCntrlCmd <> #statCntrlCmdOld AND #tempCntrlCmd <> "LPMLV30_CMD_UNDEFINED" THEN // Check if state change is requested
	          CASE #tempCntrlCmd OF // Check control command
	            "LPMLV30_CMD_UNHOLD":
	              #StateChangeInProcess := TRUE;
	              #StateRequested := "LPMLV30_STATE_EXECUTE";
	              // Check if valid state for command is in use by current mode
	              IF #statStatesInCurrentMode.unholding THEN
	                #statStateInternal := "LPMLV30_STATE_UNHOLDING";
	              ELSE
	                #statStateInternal := "LPMLV30_STATE_EXECUTE";
	              END_IF;
	            ELSE
	              IF #diagnostics.buffer[#tempDiagnosticsBufferIndexCmd].message = #MSG_NO_MESSAGE THEN // ELSE: Message was already written in head part of message handling
	                #diagnostics.buffer[#tempDiagnosticsBufferIndexCmd].message := #MSG_CMD_NOT_ALLOWED;
	              END_IF;
	          END_CASE;
	        END_IF;
	
	      "LPMLV30_STATE_SUSPENDING":
	        // Check if state is completed
	        IF #tempSCInternal AND #statStatesInCurrentMode.suspended THEN // ELSE: Wait for state complete signal
	          #statStateInternal := "LPMLV30_STATE_SUSPENDED";
	        ELSIF #tempSCInternal AND NOT #statStatesInCurrentMode.suspended THEN
	          #diagnostics.buffer[#tempDiagnosticsBufferIndexSC].message := #MSG_SC_NOT_ALLOWED;
	        END_IF;
	        
	      "LPMLV30_STATE_SUSPENDED":
	        #StateChangeInProcess := FALSE;
	        //  Check if valid command is sent
	        IF #statCmdChangeRequest AND #tempCntrlCmd <> #statCntrlCmdOld AND #tempCntrlCmd <> "LPMLV30_CMD_UNDEFINED" THEN // Check if state change is requested
	          CASE #tempCntrlCmd OF // Check control command
	            "LPMLV30_CMD_UNSUSPEND":
	              #StateChangeInProcess := TRUE;
	              #StateRequested := "LPMLV30_STATE_EXECUTE";
	              // Check if valid state for command is in use by current mode
	              IF #statStatesInCurrentMode.unsuspending THEN
	                #statStateInternal := "LPMLV30_STATE_UNSUSPENDING";
	              ELSE
	                #statStateInternal := "LPMLV30_STATE_EXECUTE";
	              END_IF;
	            ELSE
	              IF #diagnostics.buffer[#tempDiagnosticsBufferIndexCmd].message = #MSG_NO_MESSAGE THEN // ELSE: Message was already written in head part of message handling
	                #diagnostics.buffer[#tempDiagnosticsBufferIndexCmd].message := #MSG_CMD_NOT_ALLOWED;
	              END_IF;
	          END_CASE;
	        END_IF;
	        
	      "LPMLV30_STATE_ABORTING":
	        // Check if state is completed
	        IF #tempSCInternal THEN // ELSE: Wait for state complete signal
	          #statStateInternal := "LPMLV30_STATE_ABORTED";
	        END_IF;
	
	      "LPMLV30_STATE_ABORTED":
	        #StateChangeInProcess := FALSE;
	        //  Check if valid command is sent
	        IF #statCmdChangeRequest AND #tempCntrlCmd <> #statCntrlCmdOld AND #tempCntrlCmd <> "LPMLV30_CMD_UNDEFINED" THEN // Check if state change is requested
	          CASE #tempCntrlCmd OF // Check control command
	            "LPMLV30_CMD_CLEAR":
	              #StateChangeInProcess := TRUE;
	              #StateRequested := "LPMLV30_STATE_STOPPED";
	              // Check if valid state for command is in use by current mode
	              IF #statStatesInCurrentMode.clearing THEN
	                #statStateInternal := "LPMLV30_STATE_CLEARING";
	              ELSE
	                #statStateInternal := "LPMLV30_STATE_STOPPED";
	              END_IF;
	            ELSE
	              IF #diagnostics.buffer[#tempDiagnosticsBufferIndexCmd].message = #MSG_NO_MESSAGE THEN // ELSE: Message was already written in head part of message handling
	                #diagnostics.buffer[#tempDiagnosticsBufferIndexCmd].message := #MSG_CMD_NOT_ALLOWED;
	              END_IF;
	          END_CASE;
	        END_IF;
	
	      "LPMLV30_STATE_CLEARING",
	      "LPMLV30_STATE_STOPPING":
	        // Check if state is completed
	        IF #tempSCInternal THEN // ELSE: Wait for state complete signal
	          #statStateInternal := "LPMLV30_STATE_STOPPED";
	        END_IF;
	        
	      "LPMLV30_STATE_STOPPED":
	        #StateChangeInProcess := FALSE;
	        IF #statCmdChangeRequest AND #tempCntrlCmd <> #statCntrlCmdOld AND #tempCntrlCmd <> "LPMLV30_CMD_UNDEFINED" THEN // Check if state change is requested
	          // Check if valid command is sent
	          CASE #tempCntrlCmd OF
	            "LPMLV30_CMD_RESET":
	              // Check if valid state for command is in use by current unit mode
	              IF #statStatesInCurrentMode.resetting THEN
	                #StateChangeInProcess := TRUE;
	                #StateRequested    := "LPMLV30_STATE_IDLE";
	                #statStateInternal := "LPMLV30_STATE_RESETTING";
	              ELSIF #statStatesInCurrentMode.idle THEN
	                #StateChangeInProcess := TRUE;
	                #StateRequested    := "LPMLV30_STATE_IDLE";
	                #statStateInternal := "LPMLV30_STATE_IDLE";
	              ELSE
	                #diagnostics.buffer[#tempDiagnosticsBufferIndexCmd].message := #MSG_CMD_NOT_ALLOWED;
	              END_IF;
	              
	            "LPMLV30_CMD_START":
	              IF NOT #statStatesInCurrentMode.resetting AND NOT #statStatesInCurrentMode.idle THEN
	                #StateChangeInProcess := TRUE;
	                #StateRequested := "LPMLV30_STATE_EXECUTE";
	                // Check if valid state for command is in use by current mode
	                IF #statStatesInCurrentMode.starting THEN
	                  #statStateInternal := "LPMLV30_STATE_STARTING";
	                ELSE
	                  #statStateInternal := "LPMLV30_STATE_EXECUTE";
	                END_IF;
	              ELSE
	                #diagnostics.buffer[#tempDiagnosticsBufferIndexCmd].message := #MSG_CMD_NOT_ALLOWED;
	              END_IF;
	            ELSE
	              IF #diagnostics.buffer[#tempDiagnosticsBufferIndexCmd].message = #MSG_NO_MESSAGE THEN // ELSE: Message was already written in head part of message handling
	                #diagnostics.buffer[#tempDiagnosticsBufferIndexCmd].message := #MSG_CMD_NOT_ALLOWED;
	              END_IF;
	          END_CASE;
	        END_IF;
	        
	      "LPMLV30_STATE_UNDEFINED":
	        #StateChangeInProcess := FALSE;
	        #StateRequested    := "LPMLV30_STATE_STOPPED";
	        #statStateInternal := "LPMLV30_STATE_STOPPED";
	      ELSE
	        ; // Undefined state
	    END_CASE;
	  END_IF; // End: state machine
	
	  //-------------------------------------------------
	  // Message handling for state manager: foot part
	  //-------------------------------------------------
	  IF #statStateInternal <> #statStateCurrentOld THEN // ELSE: States were not changed
	    IF #tempDiagnosticsBufferIndexCmd >= 0 AND #tempDiagnosticsBufferIndexCmd <= "LPMLV30_DIAG_BUFFER_UPPER_LIM" THEN
	      IF #diagnostics.buffer[#tempDiagnosticsBufferIndexCmd].message = #MSG_NO_MESSAGE THEN
	        #diagnostics.buffer[#tempDiagnosticsBufferIndexCmd].message := #MSG_STATE_CHANGED_SUCCESSFULLY;
	      END_IF;
	    END_IF;
	    IF #tempDiagnosticsBufferIndexSC >= 0 AND #tempDiagnosticsBufferIndexSC <= "LPMLV30_DIAG_BUFFER_UPPER_LIM" THEN
	      IF #diagnostics.buffer[#tempDiagnosticsBufferIndexSC].message = #MSG_NO_MESSAGE THEN
	        #diagnostics.buffer[#tempDiagnosticsBufferIndexSC].message := #MSG_STATE_CHANGED_SUCCESSFULLY;
	      END_IF;
	    END_IF;
	  END_IF; // End: message handling for state manager: foot part
	END_IF; // End: As from second cycle
	// End: State manager
	
	//--------------------------------------------------------------------------------------------------
	// Write outputs including boolean interface outputs 
	//--------------------------------------------------------------------------------------------------
	IF #statUnitModeCurrentInternal <> #statUnitModeCurrentInternalOld THEN // Check if new unit mode is selected
	  #ProductionModeActive  := FALSE;
	  #MaintenanceModeActive := FALSE;
	  #ManualModeActive      := FALSE;
	  #UserMode01Active      := FALSE;
	  #UserMode02Active      := FALSE;
	  #UserMode03Active      := FALSE;
	  #UserMode04Active      := FALSE;
	  #UserMode05Active      := FALSE;
	  #UserMode06Active      := FALSE;
	  #UserMode07Active      := FALSE;
	  #UserMode08Active      := FALSE;
	  // #UserMode09Active := FALSE;
	  // #UserMode10Active := FALSE;
	  // #UserMode11Active := FALSE;
	  // #UserMode13Active := FALSE;
	  // #UserMode14Active := FALSE;
	  // #UserMode15Active := FALSE;
	  // #UserMode16Active := FALSE;
	  // #UserMode17Active := FALSE;
	  // #UserMode18Active := FALSE;
	  // #UserMode19Active := FALSE;
	  // #UserMode20Active := FALSE;
	  // #UserMode21Active := FALSE;
	  // #UserMode22Active := FALSE;
	  // #UserMode23Active := FALSE;
	  // #UserMode24Active := FALSE;
	  // #UserMode25Active := FALSE;
	  // #UserMode26Active := FALSE;
	  // #UserMode27Active := FALSE;
	  // #UserMode28Active := FALSE;
	
	  CASE #statUnitModeCurrentInternal OF // Set new bit for current unit mode
	    "LPMLV30_MODE_PRODUCTION":
	      #ProductionModeActive := TRUE;
	    "LPMLV30_MODE_MAINTENANCE":
	      #MaintenanceModeActive := TRUE;
	    "LPMLV30_MODE_MANUAL":
	      #ManualModeActive := TRUE;
	    "LPMLV30_MODE_USER_01":
	      #UserMode01Active := TRUE;
	    "LPMLV30_MODE_USER_02":
	      #UserMode02Active := TRUE;
	    "LPMLV30_MODE_USER_03":
	      #UserMode03Active := TRUE;
	    "LPMLV30_MODE_USER_04":
	      #UserMode04Active := TRUE;
	    "LPMLV30_MODE_USER_05":
	      #UserMode05Active := TRUE;
	    "LPMLV30_MODE_USER_06":
	      #UserMode06Active := TRUE;
	    "LPMLV30_MODE_USER_07":
	      #UserMode07Active := TRUE;
	    "LPMLV30_MODE_USER_08":
	      #UserMode08Active := TRUE;
	    // LPMLV30_MODE_USER_09:
	    //   #UserMode09Active := TRUE;
	    // LPMLV30_MODE_USER_10:
	    //   #UserMode10Active := TRUE;
	    // LPMLV30_MODE_USER_11:
	    //   #UserMode11Active := TRUE;
	    // LPMLV30_MODE_USER_12:
	    //   #UserMode12Active := TRUE;
	    // LPMLV30_MODE_USER_13:
	    //   #UserMode13Active := TRUE;
	    // LPMLV30_MODE_USER_14:
	    //   #UserMode14Active := TRUE;
	    // LPMLV30_MODE_USER_15:
	    //   #UserMode15Active := TRUE;
	    // LPMLV30_MODE_USER_16:
	    //   #UserMode16Active := TRUE;
	    // LPMLV30_MODE_USER_17:
	    //   #UserMode17Active := TRUE;
	    // LPMLV30_MODE_USER_18:
	    //   #UserMode18Active := TRUE;
	    // LPMLV30_MODE_USER_19:
	    //   #UserMode19Active := TRUE;
	    // LPMLV30_MODE_USER_20:
	    //   #UserMode20Active := TRUE;
	    // LPMLV30_MODE_USER_21:
	    //   #UserMode21Active := TRUE;
	    // LPMLV30_MODE_USER_22:
	    //   #UserMode22Active := TRUE;
	    // LPMLV30_MODE_USER_23:
	    //   #UserMode23Active := TRUE;
	    // LPMLV30_MODE_USER_24:
	    //   #UserMode25Active := TRUE;
	    // LPMLV30_MODE_USER_25:
	    //   #UserMode25Active := TRUE;
	    // LPMLV30_MODE_USER_26:
	    //   #UserMode26Active := TRUE;
	    // LPMLV30_MODE_USER_27:
	    //   #UserMode27Active := TRUE;
	    // LPMLV30_MODE_USER_28:
	    //   #UserMode28Active := TRUE;
	    ELSE
	      ; // No bit is set
	  END_CASE;
	  
	  #statUnitModeCurrentInternalOld := #statUnitModeCurrentInternal;
	END_IF;
	
	IF #statStateInternal <> #statStateInternalOld THEN // Check if new state is selected 
	  #StateCurrent := #statStateInternal; // Set output
	  
	  // Set states of boolean interface out
	  // Delete old state  
	  #ClearingStateActive     := FALSE;
	  #StoppedStateActive      := FALSE;
	  #StartingStateActive     := FALSE;
	  #IdleStateActive         := FALSE;
	  #SuspendedStateActive    := FALSE;
	  #ExecuteStateActive      := FALSE;
	  #StoppingStateActive     := FALSE;
	  #AbortingStateActive     := FALSE;
	  #AbortedStateActive      := FALSE;
	  #HoldingStateActive      := FALSE;
	  #HeldStateActive         := FALSE;
	  #UnholdingStateActive    := FALSE;
	  #SuspendingStateActive   := FALSE;
	  #UnsuspendingStateActive := FALSE;
	  #ResettingStateActive    := FALSE;
	  #CompletingStateActive   := FALSE;
	  #CompleteStateActive     := FALSE;
	
	  // Set new state
	  CASE #statStateInternal OF
	    "LPMLV30_STATE_CLEARING":
	      #ClearingStateActive := TRUE;
	    "LPMLV30_STATE_STOPPED":
	      #StoppedStateActive := TRUE;
	    "LPMLV30_STATE_STARTING":
	      #StartingStateActive := TRUE;
	    "LPMLV30_STATE_IDLE":
	      #IdleStateActive := TRUE;
	    "LPMLV30_STATE_SUSPENDED":
	      #SuspendedStateActive := TRUE;
	    "LPMLV30_STATE_EXECUTE":
	      #ExecuteStateActive := TRUE;
	    "LPMLV30_STATE_STOPPING":
	      #StoppingStateActive := TRUE;
	    "LPMLV30_STATE_ABORTING":
	      #AbortingStateActive := TRUE;
	    "LPMLV30_STATE_ABORTED":
	      #AbortedStateActive := TRUE;
	    "LPMLV30_STATE_HOLDING":
	      #HoldingStateActive := TRUE;
	    "LPMLV30_STATE_HELD":
	      #HeldStateActive := TRUE;
	    "LPMLV30_STATE_UNHOLDING":
	      #UnholdingStateActive := TRUE;
	    "LPMLV30_STATE_SUSPENDING":
	      #SuspendingStateActive := TRUE;
	    "LPMLV30_STATE_UNSUSPENDING":
	      #UnsuspendingStateActive := TRUE;
	    "LPMLV30_STATE_RESETTING":
	      #ResettingStateActive := TRUE;
	    "LPMLV30_STATE_COMPLETING":
	      #CompletingStateActive := TRUE;
	    "LPMLV30_STATE_COMPLETE":
	      #CompleteStateActive := TRUE;
	    ELSE
	      ;
	  END_CASE; // End: Set new state
	  
	  #statStateInternalOld := #statStateInternal;
	END_IF;// End: Write boolean interface outputs
	
	#diagnostics.bufferIndex := #tempDiagnosticsBufferIndex; // Temporary variable is used during block execution -> Copy back/Set output
	IF #statFirstCycle THEN
	  #statFirstCycle := FALSE;
	END_IF;
	
	// Save values for edge detection
	IF #statUnitModeChangeRequest THEN
	  #statUnitModeOld := #statUnitMode;
	END_IF;
	IF #statCmdChangeRequest THEN
	  #statCntrlCmdOld := #tempCntrlCmd;
	END_IF;
	IF #statStateInternal <> #statStateCurrentOld THEN
	  #statStateCurrentOld := #statStateInternal;
	END_IF;
	
	//============================================================================================================
	// End of function block: LPMLV30_UnitModeStateManager
	//============================================================================================================
END_FUNCTION_BLOCK

FUNCTION_BLOCK "LPMLV30_UnitModeStateTimes"
TITLE = LPMLV30_UnitModeStateTimes
{ S7_Optimized_Access := 'TRUE' }
AUTHOR : APC_ERLF
FAMILY : OMAC
//Support: tech.team.motioncontrol@siemens.com 
//Fax: +49 (0) 9131/98-1297
   VAR_INPUT 
      UnitModeCurrent : DInt := "LPMLV30_MODE_INVALID";   // Current unit mode
      StateCurrent : DInt := "LPMLV30_STATE_UNDEFINED";   // Current state
      resetTimes : Bool := false;   // State change from FALSE to TRUE (rising edge) resets unit mode/state times and cumulative times
   END_VAR

   VAR_OUTPUT 
      ModeCurrentTime : Array[0.."LPMLV30_MODES_UPPER_LIM"] of DInt;   // Current time for all modes in seconds
   END_VAR
   VAR_OUTPUT RETAIN
      ModeCumulativeTime : Array[0.."LPMLV30_MODES_UPPER_LIM"] of DInt;   // Cumulative time for all modes in seconds
   END_VAR
   VAR_OUTPUT 
      StateCurrentTime : Array[0.."LPMLV30_MODES_UPPER_LIM", 0.."LPMLV30_STATES_UPPER_LIM"] of DInt;   // Current time for all states in seconds
   END_VAR
   VAR_OUTPUT RETAIN
      StateCumulativeTime : Array[0.."LPMLV30_MODES_UPPER_LIM", 0.."LPMLV30_STATES_UPPER_LIM"] of DInt;   // Cumulative time for all states in seconds
   END_VAR
   VAR_OUTPUT 
      actualTimeCurrentMode : DInt;   // Actual time for current mode in seconds
      cumulativeTimeCurrentMode : DInt;   // Cumulative time for current mode in seconds
      actualTimeCurrentStates : Array[0.."LPMLV30_STATES_UPPER_LIM"] of DInt;   // Actual time for all states in current mode in seconds
      cumulativeTimeCurrentStates : Array[0.."LPMLV30_STATES_UPPER_LIM"] of DInt;   // Cumulative time for all states in current mode in seconds
   END_VAR
   VAR_OUTPUT RETAIN
      AccTimeSinceReset : DInt;   // Accumulated time since last reset in seconds
   END_VAR

   VAR 
      statUnitModeCurrentOld { ExternalAccessible := 'False'; ExternalVisible := 'False'; ExternalWritable := 'False'} : DInt := "LPMLV30_MODE_INVALID";   // For edge detection
      statStateCurrentOld { ExternalAccessible := 'False'; ExternalVisible := 'False'; ExternalWritable := 'False'} : DInt := "LPMLV30_STATE_UNDEFINED";   // For edge detection
      statResetTimesOld { ExternalAccessible := 'False'; ExternalVisible := 'False'; ExternalWritable := 'False'} : Bool := false;   // For edge detection
      statStartingPointMeasureRuntime { ExternalAccessible := 'False'; ExternalVisible := 'False'; ExternalWritable := 'False'} : LReal := 0.0;   // Saved value of runtime system function
      statRuntime { ExternalAccessible := 'False'; ExternalVisible := 'False'; ExternalWritable := 'False'} : LReal := 0.0;   // Runtime variable
      statFirstCycle { ExternalAccessible := 'False'; ExternalVisible := 'False'; ExternalWritable := 'False'} : Bool := true;   // First cycle of run
   END_VAR

   VAR_TEMP 
      tempI : Int;   // Loop counter
      tempJ : Int;   // Loop counter
      tempMeasuredRuntime : LReal;   // Return value of RUNTIME instruction
      tempRuntimeIntegerPart : DInt;   // Runtime variable (integer part)
      tempUnitModeCurrent : DInt;   // Verified input value
      tempStateCurrent : DInt;   // Verified input value
   END_VAR


BEGIN
	//============================================================================================================
	// SIEMENS AG
	// (c)Copyright 2015 All Rights Reserved
	//------------------------------------------------------------------------------------------------------------
	// Library: LPMLV30
	// Tested with: S7-1200 with FW version V4.1, S7-1500 with FW version V1.7
	// Engineering: TIA Portal V13 SP1
	// Restrictions: ---
	// Requirements: S7-1200 / S7-1500
	// Functionality: Determination of unit modes and states times (current and also cumulative times)
	//------------------------------------------------------------------------------------------------------------
	// Change log table:
	// Version  Date        Expert in charge    Changes applied
	// 03.00.01 29.05.2015  RK                  First released version 
	//============================================================================================================
	// Function block: LPMLV30_UnitModeStateTimes
	//============================================================================================================
	
	IF #statFirstCycle OR (#resetTimes AND NOT #statResetTimesOld) THEN
	  // Reset times structures
	  FOR #tempI := "LPMLV30_MODE_INVALID" TO "LPMLV30_MODES_UPPER_LIM" DO
	    #ModeCurrentTime[#tempI] := 0;
	    IF NOT #statFirstCycle THEN // Do only with rising edge at resetTimes
	      #ModeCumulativeTime[#tempI] := 0;
	    END_IF;
	    FOR #tempJ := "LPMLV30_STATE_UNDEFINED" TO "LPMLV30_STATES_UPPER_LIM" DO
	      #StateCurrentTime[#tempI, #tempJ] := 0;
	      IF NOT #statFirstCycle THEN // Do only with rising edge at resetTimes
	        #StateCumulativeTime[#tempI, #tempJ] := 0;
	      END_IF;
	    END_FOR;
	  END_FOR;
	  IF NOT #statFirstCycle THEN // Do only with rising edge at resetTimes
	    #AccTimeSinceReset := 0;
	  END_IF;
	  
	  // Reset additional outputs
	  #actualTimeCurrentMode := 0;
	  IF NOT #statFirstCycle THEN // Do only with rising edge at resetTimes
	    #cumulativeTimeCurrentMode := 0;
	  END_IF;
	  FOR #tempI := "LPMLV30_STATE_UNDEFINED" TO "LPMLV30_STATES_UPPER_LIM" DO
	    #actualTimeCurrentStates[#tempI] := 0;
	    IF NOT #statFirstCycle THEN // Do only with rising edge at resetTimes
	      #cumulativeTimeCurrentStates[#tempI] := 0;
	    END_IF;
	  END_FOR;
	  
	  // Set starting point for calculation of elapsed seconds
	  #tempMeasuredRuntime := RUNTIME(#statStartingPointMeasureRuntime);
	  #statRuntime := 0.0;
	  
	  IF #statFirstCycle THEN
	    #statFirstCycle := FALSE;
	    RETURN; // Nothing else in this cycle to avoid runtime peaks
	  END_IF;
	END_IF;
	
	// Inputs UnitModeCurrent and StateCurrent
	#tempUnitModeCurrent := #UnitModeCurrent;
	#tempStateCurrent    := #StateCurrent;
	
	// Measure program runtime
	#tempMeasuredRuntime := RUNTIME(#statStartingPointMeasureRuntime);
	IF #tempMeasuredRuntime > 0.0 THEN //value OK
	  #statRuntime := #statRuntime + #tempMeasuredRuntime;
	END_IF;
	
	// Check if at least one second has been reached
	IF #statRuntime > 1.0 THEN
	  #tempRuntimeIntegerPart := TRUNC_DINT(#statRuntime);
	  
	  IF #statUnitModeCurrentOld >= "LPMLV30_MODE_INVALID" AND #statUnitModeCurrentOld <= "LPMLV30_MODES_UPPER_LIM" THEN
	    //DINT overflow is not taken into account, because DINT in seconds means approx. 68 years
	    #ModeCurrentTime[#statUnitModeCurrentOld]    := #ModeCurrentTime[#statUnitModeCurrentOld]    + #tempRuntimeIntegerPart;
	    #ModeCumulativeTime[#statUnitModeCurrentOld] := #ModeCumulativeTime[#statUnitModeCurrentOld] + #tempRuntimeIntegerPart;
	
	    IF #statStateCurrentOld >= "LPMLV30_STATE_UNDEFINED" AND #statStateCurrentOld <= "LPMLV30_STATES_UPPER_LIM" THEN
	      //DINT overflow is not taken into account, because DINT in seconds means approx. 68 years
	      #StateCurrentTime[#statUnitModeCurrentOld, #statStateCurrentOld]    := #StateCurrentTime[#statUnitModeCurrentOld, #statStateCurrentOld]    + #tempRuntimeIntegerPart;
	      #StateCumulativeTime[#statUnitModeCurrentOld, #statStateCurrentOld] := #StateCumulativeTime[#statUnitModeCurrentOld, #statStateCurrentOld] + #tempRuntimeIntegerPart;
	    END_IF;
	  END_IF;
	
	  //DINT overflow is not taken into account, because DINT in seconds means approx. 68 years
	  #AccTimeSinceReset := #AccTimeSinceReset + #tempRuntimeIntegerPart;
	
	  #statRuntime := #statRuntime - #tempRuntimeIntegerPart; //fractional part of runtime variable for next cycle
	END_IF;
	
	// Check if new unitMode is selected
	IF #tempUnitModeCurrent <> #statUnitModeCurrentOld THEN
	  IF #tempUnitModeCurrent >= "LPMLV30_MODE_INVALID" AND #tempUnitModeCurrent <= "LPMLV30_MODES_UPPER_LIM" THEN
	    #ModeCurrentTime[#tempUnitModeCurrent] := 0;
	    IF #tempStateCurrent >= "LPMLV30_STATE_UNDEFINED" AND #tempStateCurrent <= "LPMLV30_STATES_UPPER_LIM" THEN
	      #StateCurrentTime[#tempUnitModeCurrent, #tempStateCurrent] := 0;
	    END_IF;
	  END_IF;
	
	// Check if new state is selected   
	ELSIF #tempStateCurrent <> #statStateCurrentOld THEN
	  IF #tempUnitModeCurrent >= "LPMLV30_MODE_INVALID"    AND #tempUnitModeCurrent <= "LPMLV30_MODES_UPPER_LIM" AND
	     #tempStateCurrent    >= "LPMLV30_STATE_UNDEFINED" AND #tempStateCurrent    <= "LPMLV30_STATES_UPPER_LIM"
	  THEN
	    #StateCurrentTime[#tempUnitModeCurrent, #tempStateCurrent] := 0;
	  END_IF;
	END_IF;
	
	// Update additional outputs
	IF #tempUnitModeCurrent >= "LPMLV30_MODE_INVALID" AND #tempUnitModeCurrent <= "LPMLV30_MODES_UPPER_LIM" THEN
	  #actualTimeCurrentMode     := #ModeCurrentTime[#tempUnitModeCurrent];
	  #cumulativeTimeCurrentMode := #ModeCumulativeTime[#tempUnitModeCurrent];
	  IF #tempStateCurrent >= "LPMLV30_STATE_UNDEFINED" AND #tempStateCurrent <= "LPMLV30_STATES_UPPER_LIM" THEN
	    #actualTimeCurrentStates     := #StateCurrentTime[#tempUnitModeCurrent];
	    #cumulativeTimeCurrentStates := #StateCumulativeTime[#tempUnitModeCurrent];
	  ELSE
	    FOR #tempI := "LPMLV30_STATE_UNDEFINED" TO "LPMLV30_STATES_UPPER_LIM" DO
	      #actualTimeCurrentStates[#tempI] := 0;
	      #cumulativeTimeCurrentStates[#tempI] := 0;
	    END_FOR;
	  END_IF;
	ELSE
	  #actualTimeCurrentMode     := 0;
	  #cumulativeTimeCurrentMode := 0;
	
	  FOR #tempI := "LPMLV30_STATE_UNDEFINED" TO "LPMLV30_STATES_UPPER_LIM" DO
	    #actualTimeCurrentStates[#tempI]     := 0;
	    #cumulativeTimeCurrentStates[#tempI] := 0;
	  END_FOR;
	END_IF;
	
	// Save values for state change detection
	#statResetTimesOld      := #resetTimes;
	#statUnitModeCurrentOld := #tempUnitModeCurrent;
	#statStateCurrentOld    := #tempStateCurrent;
	
	//============================================================================================================
	// End of Function block: LPMLV30_UnitModeStateTimes
	//============================================================================================================
END_FUNCTION_BLOCK

FUNCTION "LPMLV30_GetUnitModeStateNamesAsString" : Void
TITLE = LPMLV30_GetUnitModeStateNamesAsString
{ S7_Optimized_Access := 'TRUE' }
AUTHOR : APC_ERLF
FAMILY : OMAC
//Support: tech.team.motioncontrol@siemens.com 
//Fax: +49 (0) 9131/98-1297
   VAR_INPUT 
      UnitModeCurrent : DInt;   // Current unit mode
      StateCurrent : DInt;   // Current state
      language : Int;   // Requested language (LPMLV30_LANGUAGE_1, LPMLV30_LANGUAGE_2, ...)
      namesConfiguration : "typeLPMLV30_NamesConfiguration";   // All names of unit modes and states (in different languages)
   END_VAR

   VAR_OUTPUT 
      unitModeCurrentName : String;   // Name of current unit mode in the requested language
      stateCurrentName : String;   // Name of current state in the requested language
   END_VAR

   VAR_TEMP 
      tempUnitModeCurrent : DInt;   // Current unit mode
      tempStateCurrent : DInt;   // Current state
      tempLanguage : Int;   // Requested language
   END_VAR


BEGIN
	//============================================================================================================
	// SIEMENS AG
	// (c)Copyright 2015 All Rights Reserved
	//------------------------------------------------------------------------------------------------------------
	// Library: LPMLV30
	// Tested with: S7-1200 with FW version V4.1, S7-1500 with FW version V1.7
	// Engineering: TIA Portal V13 SP1
	// Restrictions: ---
	// Requirements: S7-1200 / S7-1500
	// Functionality: Gets the names for current unit mode and state in one language 
	//                corresponding to the names configuration
	//------------------------------------------------------------------------------------------------------------
	// Change log table:
	// Version  Date        Expert in charge    Changes applied
	// 03.00.01 29.05.2015  RK                  First released version 
	//============================================================================================================
	// Function: LPMLV30_GetUnitModeStateNamesAsString
	//============================================================================================================
	
	#tempUnitModeCurrent := #UnitModeCurrent;
	#tempStateCurrent    := #StateCurrent;
	#tempLanguage        := #language;
	
	IF #tempUnitModeCurrent < 0 OR #tempUnitModeCurrent > "LPMLV30_MODES_UPPER_LIM" THEN
	  #tempUnitModeCurrent := "LPMLV30_MODE_INVALID";
	END_IF;
	IF #tempStateCurrent < 0 OR #tempStateCurrent > "LPMLV30_STATES_UPPER_LIM" THEN
	  #tempStateCurrent := "LPMLV30_STATE_UNDEFINED";
	END_IF;
	IF #tempLanguage < 0 OR #tempLanguage > "LPMLV30_LANGUAGES_UPPER_LIM" THEN
	  #tempLanguage := "LPMLV30_LANGUAGE_1";
	END_IF;
	
	#unitModeCurrentName := #namesConfiguration.unitModesNames[#tempLanguage, #tempUnitModeCurrent];
	#stateCurrentName    := #namesConfiguration.statesNames[#tempLanguage, #tempStateCurrent];
	
	//============================================================================================================
	// End of function: LPMLV30_GetUnitModeStateNamesAsString
	//============================================================================================================
END_FUNCTION

FUNCTION_BLOCK "UN_03_LineComm"   // FB31623, LAD
TITLE = UN_03_LineComm
{ S7_Optimized_Access := 'TRUE' }
AUTHOR : tech.team.motioncontrol@siemens.com
FAMILY : CPG
VERSION : 1.0
// Support: tech.team.motioncontrol@siemens.com
// Fax: +49 (0) 9131/98-1297
// stored: AutoNumber true, IsIECCheckEnabled false, IsRetainMemResEnabled false, MemoryReserve 100, SetENOAutomatically false, UDAEnableTagReadback false
   VAR
      instAlarmRemoteStop { ExternalAccessible := 'False'; ExternalVisible := 'False'; ExternalWritable := 'False'; S7_SetPoint := 'True'} : "CPG_Event";   // Remote Command - Stop
      instAlarmRemoteAbort { ExternalAccessible := 'False'; ExternalVisible := 'False'; ExternalWritable := 'False'; S7_SetPoint := 'True'} : "CPG_Event";   // Remote Command - Abort
      instAlarmRemoteSuspendBlocked { ExternalAccessible := 'False'; ExternalVisible := 'False'; ExternalWritable := 'False'; S7_SetPoint := 'True'} : "CPG_Event";   // Remote Command - Suspend (Blocked)
      instAlarmRemoteSuspendStarved { ExternalAccessible := 'False'; ExternalVisible := 'False'; ExternalWritable := 'False'; S7_SetPoint := 'True'} : "CPG_Event";   // Remote Command - Suspend (Starved)
      instAlarmRemoteHold { ExternalAccessible := 'False'; ExternalVisible := 'False'; ExternalWritable := 'False'; S7_SetPoint := 'True'} : "CPG_Event";   // Remote Command - Hold
      statRemoteSuspendCommand { ExternalAccessible := 'False'; ExternalVisible := 'False'; ExternalWritable := 'False'} : Bool;   // Remote Suspend Command is active (from remote station)
      statRemoteHoldCommand { ExternalAccessible := 'False'; ExternalVisible := 'False'; ExternalWritable := 'False'} : Bool;   // Remote Hold Command is active (from remote station)
   END_VAR
BEGIN

REGION Network 1: *** COMMUNICATION LOGIC ***
END_REGION

REGION Network 2: *** REMOTE COMMAND LOGIC ***
END_REGION

REGION Network 3: Remote Stop Command
   // "PackTags".Command.CntrlCmd = 3 (stop command value)
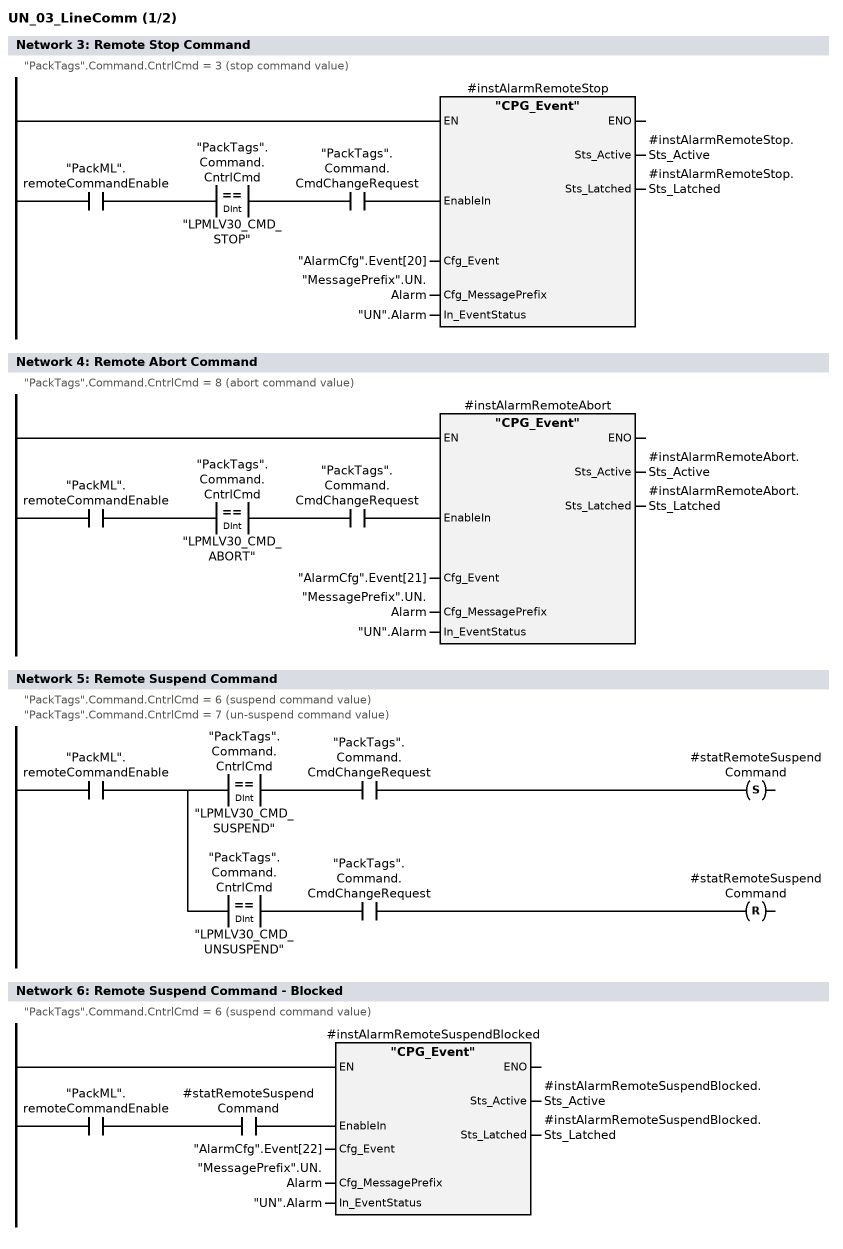
   RUNG wire#powerrail
      #instAlarmRemoteStop(EnableIn := wire#w1, Cfg_Event := "AlarmCfg".Event[20], Cfg_MessagePrefix := "MessagePrefix".UN.Alarm, In_EventStatus := "UN".Alarm, Sts_Active => #instAlarmRemoteStop.Sts_Active, Sts_Latched => #instAlarmRemoteStop.Sts_Latched)
   END_RUNG
   RUNG wire#powerrail
      Contact( "PackML".remoteCommandEnable )
      { S7_Templates := "SrcType := DInt" } EQ_Contact(in1 := "PackTags".Command.CntrlCmd, in2 := "LPMLV30_CMD_STOP")
      Contact( "PackTags".Command.CmdChangeRequest )
   END_RUNG wire#w1
   // the same network as SCL:
   #instAlarmRemoteStop(EnableIn := "PackML".remoteCommandEnable AND ("PackTags".Command.CntrlCmd = "LPMLV30_CMD_STOP") AND "PackTags".Command.CmdChangeRequest,   // "CPG_Event"
                        Cfg_Event := "AlarmCfg".Event[20],
                        Cfg_MessagePrefix := "MessagePrefix".UN.Alarm,
                        In_EventStatus := "UN".Alarm,
                        Sts_Active => #instAlarmRemoteStop.Sts_Active,
                        Sts_Latched => #instAlarmRemoteStop.Sts_Latched);
END_REGION

REGION Network 4: Remote Abort Command
   // "PackTags".Command.CntrlCmd = 8 (abort command value)
   RUNG wire#powerrail
      #instAlarmRemoteAbort(EnableIn := wire#w1, Cfg_Event := "AlarmCfg".Event[21], Cfg_MessagePrefix := "MessagePrefix".UN.Alarm, In_EventStatus := "UN".Alarm, Sts_Active => #instAlarmRemoteAbort.Sts_Active, Sts_Latched => #instAlarmRemoteAbort.Sts_Latched)
   END_RUNG
   RUNG wire#powerrail
      Contact( "PackML".remoteCommandEnable )
      { S7_Templates := "SrcType := DInt" } EQ_Contact(in1 := "PackTags".Command.CntrlCmd, in2 := "LPMLV30_CMD_ABORT")
      Contact( "PackTags".Command.CmdChangeRequest )
   END_RUNG wire#w1
   // the same network as SCL:
   #instAlarmRemoteAbort(EnableIn := "PackML".remoteCommandEnable AND ("PackTags".Command.CntrlCmd = "LPMLV30_CMD_ABORT") AND "PackTags".Command.CmdChangeRequest,   // "CPG_Event"
                         Cfg_Event := "AlarmCfg".Event[21],
                         Cfg_MessagePrefix := "MessagePrefix".UN.Alarm,
                         In_EventStatus := "UN".Alarm,
                         Sts_Active => #instAlarmRemoteAbort.Sts_Active,
                         Sts_Latched => #instAlarmRemoteAbort.Sts_Latched);
END_REGION

REGION Network 5: Remote Suspend Command
   // "PackTags".Command.CntrlCmd = 6 (suspend command value)
   // "PackTags".Command.CntrlCmd = 7 (un-suspend command value)
   RUNG wire#powerrail
      Contact( "PackML".remoteCommandEnable )
      wire#w1
      { S7_Templates := "SrcType := DInt" } EQ_Contact(in1 := "PackTags".Command.CntrlCmd, in2 := "LPMLV30_CMD_SUSPEND")
      Contact( "PackTags".Command.CmdChangeRequest )
      S_Coil( #statRemoteSuspendCommand )
   END_RUNG
   RUNG wire#w1
      { S7_Templates := "SrcType := DInt" } EQ_Contact(in1 := "PackTags".Command.CntrlCmd, in2 := "LPMLV30_CMD_UNSUSPEND")
      Contact( "PackTags".Command.CmdChangeRequest )
      R_Coil( #statRemoteSuspendCommand )
   END_RUNG
   // the same network as SCL:
   IF "PackML".remoteCommandEnable AND ("PackTags".Command.CntrlCmd = "LPMLV30_CMD_SUSPEND") AND "PackTags".Command.CmdChangeRequest THEN
       #statRemoteSuspendCommand := TRUE;
   END_IF;
   IF "PackML".remoteCommandEnable AND ("PackTags".Command.CntrlCmd = "LPMLV30_CMD_UNSUSPEND") AND "PackTags".Command.CmdChangeRequest THEN
       #statRemoteSuspendCommand := FALSE;
   END_IF;
END_REGION

REGION Network 6: Remote Suspend Command - Blocked
   // "PackTags".Command.CntrlCmd = 6 (suspend command value)
   RUNG wire#powerrail
      #instAlarmRemoteSuspendBlocked(EnableIn := wire#w1, Cfg_Event := "AlarmCfg".Event[22], Cfg_MessagePrefix := "MessagePrefix".UN.Alarm, In_EventStatus := "UN".Alarm, Sts_Active => #instAlarmRemoteSuspendBlocked.Sts_Active, Sts_Latched => #instAlarmRemoteSuspendBlocked.Sts_Latched)
   END_RUNG
   RUNG wire#powerrail
      Contact( "PackML".remoteCommandEnable )
      Contact( #statRemoteSuspendCommand )
   END_RUNG wire#w1
   // the same network as SCL:
   #instAlarmRemoteSuspendBlocked(EnableIn := "PackML".remoteCommandEnable AND #statRemoteSuspendCommand,   // "CPG_Event"
                           Cfg_Event := "AlarmCfg".Event[22],
                           Cfg_MessagePrefix := "MessagePrefix".UN.Alarm,
                           In_EventStatus := "UN".Alarm,
                           Sts_Active => #instAlarmRemoteSuspendBlocked.Sts_Active,
                           Sts_Latched => #instAlarmRemoteSuspendBlocked.Sts_Latched);
END_REGION

REGION Network 7: Remote Suspend Command - Starved
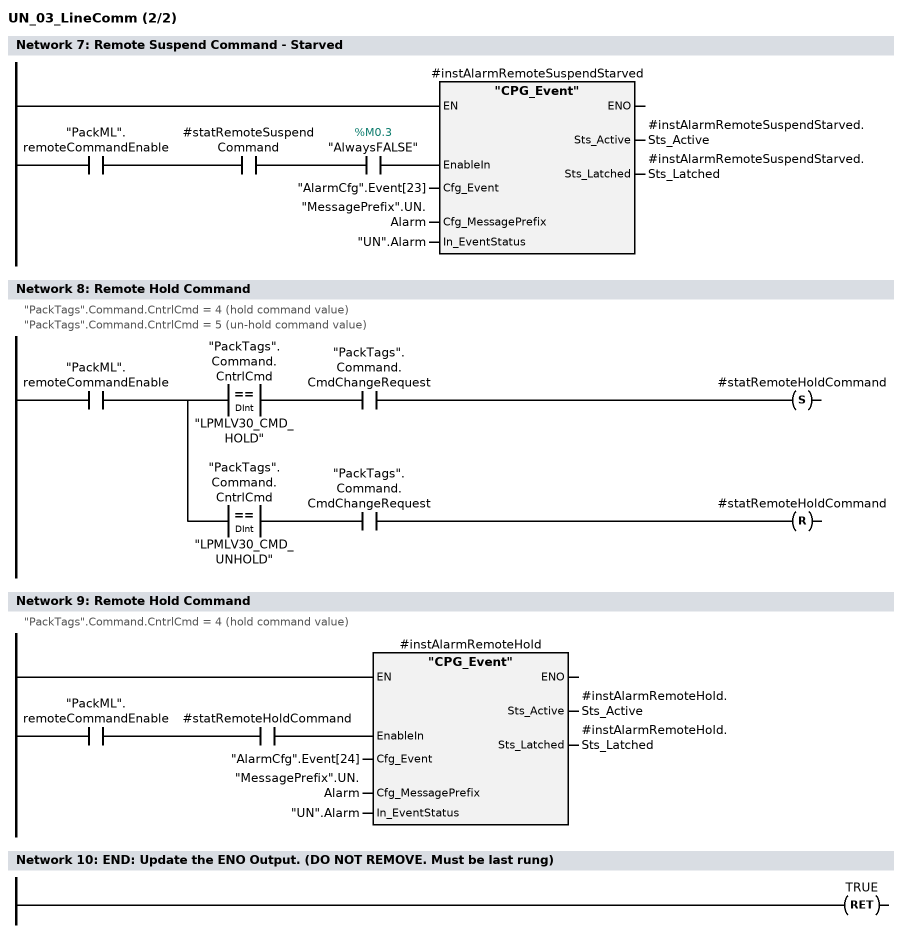
   RUNG wire#powerrail
      #instAlarmRemoteSuspendStarved(EnableIn := wire#w1, Cfg_Event := "AlarmCfg".Event[23], Cfg_MessagePrefix := "MessagePrefix".UN.Alarm, In_EventStatus := "UN".Alarm, Sts_Active => #instAlarmRemoteSuspendStarved.Sts_Active, Sts_Latched => #instAlarmRemoteSuspendStarved.Sts_Latched)
   END_RUNG
   RUNG wire#powerrail
      Contact( "PackML".remoteCommandEnable )
      Contact( #statRemoteSuspendCommand )
      Contact( "AlwaysFALSE" )
   END_RUNG wire#w1
   // the same network as SCL:
   #instAlarmRemoteSuspendStarved(EnableIn := "PackML".remoteCommandEnable AND #statRemoteSuspendCommand AND "AlwaysFALSE",   // "CPG_Event"
                           Cfg_Event := "AlarmCfg".Event[23],
                           Cfg_MessagePrefix := "MessagePrefix".UN.Alarm,
                           In_EventStatus := "UN".Alarm,
                           Sts_Active => #instAlarmRemoteSuspendStarved.Sts_Active,
                           Sts_Latched => #instAlarmRemoteSuspendStarved.Sts_Latched);
END_REGION

REGION Network 8: Remote Hold Command
   // "PackTags".Command.CntrlCmd = 4 (hold command value)
   // "PackTags".Command.CntrlCmd = 5 (un-hold command value)
   RUNG wire#powerrail
      Contact( "PackML".remoteCommandEnable )
      wire#w1
      { S7_Templates := "SrcType := DInt" } EQ_Contact(in1 := "PackTags".Command.CntrlCmd, in2 := "LPMLV30_CMD_HOLD")
      Contact( "PackTags".Command.CmdChangeRequest )
      S_Coil( #statRemoteHoldCommand )
   END_RUNG
   RUNG wire#w1
      { S7_Templates := "SrcType := DInt" } EQ_Contact(in1 := "PackTags".Command.CntrlCmd, in2 := "LPMLV30_CMD_UNHOLD")
      Contact( "PackTags".Command.CmdChangeRequest )
      R_Coil( #statRemoteHoldCommand )
   END_RUNG
   // the same network as SCL:
   IF "PackML".remoteCommandEnable AND ("PackTags".Command.CntrlCmd = "LPMLV30_CMD_HOLD") AND "PackTags".Command.CmdChangeRequest THEN
       #statRemoteHoldCommand := TRUE;
   END_IF;
   IF "PackML".remoteCommandEnable AND ("PackTags".Command.CntrlCmd = "LPMLV30_CMD_UNHOLD") AND "PackTags".Command.CmdChangeRequest THEN
       #statRemoteHoldCommand := FALSE;
   END_IF;
END_REGION

REGION Network 9: Remote Hold Command
   // "PackTags".Command.CntrlCmd = 4 (hold command value)
   RUNG wire#powerrail
      #instAlarmRemoteHold(EnableIn := wire#w1, Cfg_Event := "AlarmCfg".Event[24], Cfg_MessagePrefix := "MessagePrefix".UN.Alarm, In_EventStatus := "UN".Alarm, Sts_Active => #instAlarmRemoteHold.Sts_Active, Sts_Latched => #instAlarmRemoteHold.Sts_Latched)
   END_RUNG
   RUNG wire#powerrail
      Contact( "PackML".remoteCommandEnable )
      Contact( #statRemoteHoldCommand )
   END_RUNG wire#w1
   // the same network as SCL:
   #instAlarmRemoteHold(EnableIn := "PackML".remoteCommandEnable AND #statRemoteHoldCommand,   // "CPG_Event"
                        Cfg_Event := "AlarmCfg".Event[24],
                        Cfg_MessagePrefix := "MessagePrefix".UN.Alarm,
                        In_EventStatus := "UN".Alarm,
                        Sts_Active => #instAlarmRemoteHold.Sts_Active,
                        Sts_Latched => #instAlarmRemoteHold.Sts_Latched);
END_REGION

REGION Network 10: END: Update the ENO Output. (DO NOT REMOVE. Must be last rung)
   RUNG wire#powerrail
      ReturnCoil( TRUE )
   END_RUNG
   // the same network as SCL:
   ENO := TRUE;
   RETURN;
END_REGION
END_FUNCTION_BLOCK

FUNCTION_BLOCK "CPG_Event"
TITLE = CPG_Event
{ S7_Optimized_Access := 'TRUE' }
AUTHOR : 'tech.team.motioncontrol@siemens.com'
FAMILY : CPG
VERSION : 1.1
//Support: tech.team.motioncontrol@siemens.com
   VAR_INPUT 
      EnableIn { ExternalAccessible := 'False'; ExternalVisible := 'False'; ExternalWritable := 'False'} : Bool;   // Enable the FB call.
      Cfg_Event { ExternalAccessible := 'False'; ExternalVisible := 'False'; ExternalWritable := 'False'} : "CPG_typeEventCfg";   // configuration data structure for this event
      Cfg_MessagePrefix { ExternalAccessible := 'False'; ExternalVisible := 'False'; ExternalWritable := 'False'} : "CPG_typeMessagePrefix";   // Message Prefix value for event messages
   END_VAR

   VAR_OUTPUT 
      Sts_Active { ExternalAccessible := 'False'; ExternalVisible := 'False'; ExternalWritable := 'False'} : Bool;   // event is currently active
      Sts_Latched { ExternalAccessible := 'False'; ExternalVisible := 'False'; ExternalWritable := 'False'} : Bool;   // event has been active since last reset command
   END_VAR

   VAR_IN_OUT 
      In_EventStatus : "CPG_typeEventStatus";   // Working event list data section
   END_VAR

   VAR 
      statActive : Bool;   // event is currently active
      statLatched : Bool;   // event has been active since last reset command
      statEvent_Number { ExternalAccessible := 'False'; ExternalVisible := 'False'; ExternalWritable := 'False'} : Int;   // Event Number
      statPrev_ResetID { ExternalAccessible := 'False'; ExternalVisible := 'False'; ExternalWritable := 'False'} : Int;   // Prev Reset ID
      statError_RTC { ExternalAccessible := 'False'; ExternalVisible := 'False'; ExternalWritable := 'False'} : Int;   // Error code for reading of Real Time Clock
      statEvent_CurDateTime {InstructionName := 'DTL'; LibVersion := '1.0'; ExternalAccessible := 'False'; ExternalVisible := 'False'; ExternalWritable := 'False'} : DTL;   // temp value for current date & time
   END_VAR

   VAR_TEMP 
      tempLanguage : Int;   // value of the currently selected language
   END_VAR


BEGIN
	//============================================================================================================
	// SIEMENS AG
	// (c)Copyright 2018 All Rights Reserved
	//------------------------------------------------------------------------------------------------------------
	// Project: CPG Template
	// Tested with: S7-1500 with FW version V2.1
	// Engineering: TIA Portal V14
	// Restrictions: ---
	// Requirements: S7-1500
	// Functionality: Control TR88 EVENT functions for CPG Template. 
	// Support: tech.team.motioncontrol@siemens.com
	//------------------------------------------------------------------------------------------------------------
	// Change log table:
	// Version       Date               Expert in charge    Changes applied
	//  01.00.00     01.01.2018         MP                  Initial Release & PackML V1.8  Renamed CPG V1.0
	//  01.01.00     22.05.2018         JP                  Adopted to styleguide
	//  01.01.01     06.02.2020         KB                  Optimized call of Concat instruction
	//                                                      Changed RD_SYS_T -> RD_LOC_T
	//============================================================================================================
	// Function : CPG_Event
	//============================================================================================================
	
	// ===========================================================================
	//  Begin the LOGIC section:
	
	//-------------  If ENABLE is FALSE----------------------------------------
	IF NOT (#EnableIn) THEN                          // If block is not enabled, then
	  IF #statActive THEN              // Status Active
	    IF #statEvent_Number < #In_EventStatus.wrk_EventArraySize THEN   // current event below max size?
	      #statError_RTC := RD_LOC_T(#statEvent_CurDateTime);            // Read the Real Time Clock
	      #In_EventStatus.sts_Events[#statEvent_Number].AckDateTimeDTL := #statEvent_CurDateTime; // update Acknowledge time
	      #In_EventStatus.sts_Events[#statEvent_Number].Trigger := FALSE;
	    END_IF;                     // IF Event_Number
	
	    #statActive := FALSE;             // Reset the active bit        
	    #In_EventStatus.wrk_UpdateEventListID := #In_EventStatus.wrk_UpdateEventListID + 1;
	  END_IF;                             // IF Sts_Active
	
	  IF #statLatched AND (#In_EventStatus.wrk_ResetID <> #statPrev_ResetID) THEN
	    #statLatched := FALSE;
	    #In_EventStatus.wrk_UpdateEventListID := #In_EventStatus.wrk_UpdateEventListID + 1;
	    #statPrev_ResetID := #In_EventStatus.wrk_ResetID;
	  END_IF;             // IF Sts_Latched
	
	  ENO := FALSE;         // enable out is false (0)
	
	ELSE                    // else IF NOT (enable)
	  //-------------  If ENABLE is TRUE ----------------------------------------  
	  // If this FB is enabled....  
	  IF NOT (#statActive) OR (#In_EventStatus.wrk_ResetID <> #statPrev_ResetID) THEN
	    IF NOT (#statLatched) THEN
	      #statError_RTC := RD_LOC_T(#statEvent_CurDateTime);            // Read the Real Time Clock
	    END_IF;
	
	    IF NOT (#statLatched) OR (#In_EventStatus.wrk_ResetID <> #statPrev_ResetID) THEN
	      #statEvent_Number := #In_EventStatus.sts_NumAllEvents;             // increment event number
	      #In_EventStatus.sts_NumAllEvents := #In_EventStatus.sts_NumAllEvents + 1;         // increment number of all event
	      #statPrev_ResetID := #In_EventStatus.wrk_ResetID;                                     // update previous Reset ID      
	    END_IF;
	
	    IF #statEvent_Number < #In_EventStatus.wrk_EventArraySize THEN
	      #tempLanguage := #In_EventStatus.wrk_LanguageSelection;
	
	      #In_EventStatus.sts_Events[#statEvent_Number].ID := #Cfg_Event.ID;
	      #In_EventStatus.sts_Events[#statEvent_Number].Value := #Cfg_Event.value;
	      #In_EventStatus.sts_Events[#statEvent_Number].Category := #Cfg_Event.category;
	
	      // update the event message String with "UN"/EM prefix + CM prefix + event message for selected language
	      IF #tempLanguage >= 0 AND #tempLanguage <= "LPMLV30_LANGUAGES_UPPER_LIM" THEN
	          #In_EventStatus.sts_Events[#statEvent_Number].Message := CONCAT(IN1 := #In_EventStatus.wrk_MessagePrefix,
	                                                                          IN2 := #Cfg_MessagePrefix.messagePrefix[#tempLanguage], IN3 := #Cfg_Event.message[#tempLanguage]);
	      ELSE
	          #In_EventStatus.sts_Events[#statEvent_Number].Message := #In_EventStatus.wrk_MessagePrefix;
	      END_IF;
	      
	      
	      #In_EventStatus.sts_Events[#statEvent_Number].Trigger := TRUE;                          // Set trigger to 1 
	      #In_EventStatus.sts_Events[#statEvent_Number].DateTimeDTL := #statEvent_CurDateTime;       // Update with the current time
	      #In_EventStatus.sts_Events[#statEvent_Number].AckDateTimeDTL := DT#1990-1-1-0:0:0.0;       // clear the acknowledge time value 
	    END_IF;
	
	    #statActive := TRUE;                            // set the status active bit
	    #statLatched := TRUE;                            // set the status latched bit
	    #In_EventStatus.wrk_UpdateEventListID := #In_EventStatus.wrk_UpdateEventListID + 1;  // increment the work update listID
	
	    CASE DINT_TO_INT(#Cfg_Event.category) OF                     // set the appropriate category lateched bit
	      0:
	        #In_EventStatus.sts_Category_0_Latched := TRUE;
	      1:
	        #In_EventStatus.sts_Category_1_Latched := TRUE;
	      2:
	        #In_EventStatus.sts_Category_2_Latched := TRUE;
	      3:
	        #In_EventStatus.sts_Category_3_Latched := TRUE;
	      4:
	        #In_EventStatus.sts_Category_4_Latched := TRUE;
	      5:
	        #In_EventStatus.sts_Category_5_Latched := TRUE;
	      6:
	        #In_EventStatus.sts_Category_6_Latched := TRUE;
	      7:
	        #In_EventStatus.sts_Category_7_Latched := TRUE;
	      8:
	        #In_EventStatus.sts_Category_8_Latched := TRUE;
	      9:
	        #In_EventStatus.sts_Category_9_Latched := TRUE;
	    END_CASE;
	  END_IF; // End "IF NOT (Sts_Active)"
	
	END_IF; // End "IF NOT(EnableIn) "
	
	// Write output variables
	#Sts_Latched := #statLatched;
	#Sts_Active := #statActive;
	
	//  -------------- END OF LOGIC -------------------------
	ENO := TRUE;   // Set the ENO output
END_FUNCTION_BLOCK

FUNCTION_BLOCK "UN_04_EventControl"   // FB31624, LAD
TITLE = UN_04_EventControl
{ S7_Optimized_Access := 'TRUE' }
AUTHOR : tech.team.motioncontrol@siemens.com
FAMILY : CPG
VERSION : 1.1
// Support: tech.team.motioncontrol@siemens.com
// stored: AutoNumber true, IsIECCheckEnabled false, IsRetainMemResEnabled false, MemoryReserve 100, SetENOAutomatically false, UDAEnableTagReadback false
   VAR
      instEventMgrAlarm { ExternalAccessible := 'False'; ExternalVisible := 'False'; ExternalWritable := 'False'; S7_SetPoint := 'True'} : "CPG_EventManager";   // instance FB - Event Manager - Alarms Events
      instEventMgrWarning { ExternalAccessible := 'False'; ExternalVisible := 'False'; ExternalWritable := 'False'; S7_SetPoint := 'True'} : "CPG_EventManager";   // instance FB - Event Manager - Warning Events
      instEventMgrStatus { ExternalAccessible := 'False'; ExternalVisible := 'False'; ExternalWritable := 'False'; S7_SetPoint := 'True'} : "CPG_EventManager";   // instance FB - Event Manager - Status Events
      instStatusAlarmsNotReset { ExternalAccessible := 'False'; ExternalVisible := 'False'; ExternalWritable := 'False'; S7_SetPoint := 'True'} : "CPG_Event";   // Status = Alarms Not Reset
      statEventMgr_Cmd_Reset { ExternalAccessible := 'False'; ExternalVisible := 'False'; ExternalWritable := 'False'} : Bool;   // Reset Cmd for event managers
      statEventMgr_Cmd_Clear1stFlt { ExternalAccessible := 'False'; ExternalVisible := 'False'; ExternalWritable := 'False'} : Bool;   // Clear 1st Fault Cmd for event managers
      statEventMgr_Clear1stFlt_OS { ExternalAccessible := 'False'; ExternalVisible := 'False'; ExternalWritable := 'False'} : Bool;   // Clear 1st Fault Cmd - One shot
   END_VAR
   VAR_TEMP   // added for the SCL form of the ladder/FBD networks
      _w1 : Bool;
      _w2 : Bool;
   END_VAR
BEGIN

REGION Network 2: ** STATE MODEL REPORTING STATUS ****
END_REGION

REGION Network 3: *** Call the PackML Module Initialize Logic ***
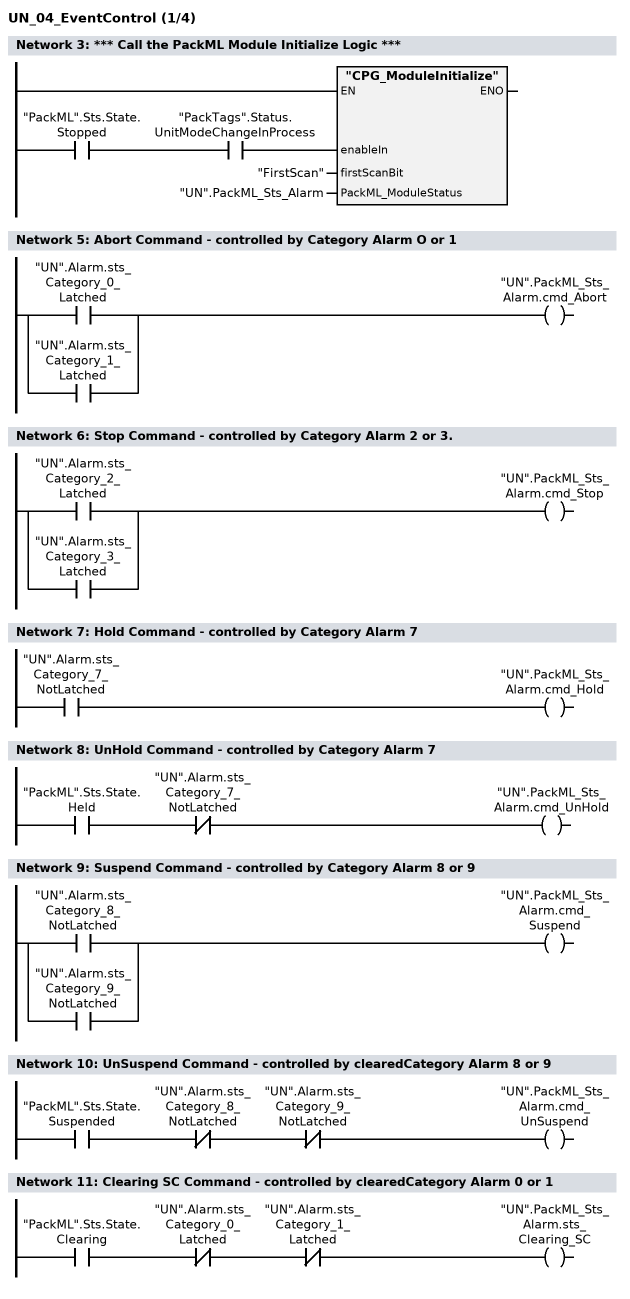
   RUNG wire#powerrail
      "CPG_ModuleInitialize"(enableIn := wire#w1, firstScanBit := "FirstScan", PackML_ModuleStatus := "UN".PackML_Sts_Alarm)
   END_RUNG
   RUNG wire#powerrail
      Contact( "PackML".Sts.State.Stopped )
      Contact( "PackTags".Status.UnitModeChangeInProcess )
   END_RUNG wire#w1
   // the same network as SCL:
   "CPG_ModuleInitialize"(enableIn := "PackML".Sts.State.Stopped AND "PackTags".Status.UnitModeChangeInProcess,
                          firstScanBit := "FirstScan",
                          PackML_ModuleStatus := "UN".PackML_Sts_Alarm);
END_REGION

REGION Network 4: Begin the LOGIC section.
END_REGION

REGION Network 5: Abort Command - controlled by Category Alarm O or 1
   RUNG wire#powerrail
      Contact( "UN".Alarm.sts_Category_0_Latched )
      wire#w1
      Coil( "UN".PackML_Sts_Alarm.cmd_Abort )
   END_RUNG
   RUNG wire#powerrail
      Contact( "UN".Alarm.sts_Category_1_Latched )
   END_RUNG wire#w1
   // the same network as SCL:
   "UN".PackML_Sts_Alarm.cmd_Abort := "UN".Alarm.sts_Category_0_Latched OR "UN".Alarm.sts_Category_1_Latched;
END_REGION

REGION Network 6: Stop Command - controlled by Category Alarm 2 or 3.
   RUNG wire#powerrail
      Contact( "UN".Alarm.sts_Category_2_Latched )
      wire#w1
      Coil( "UN".PackML_Sts_Alarm.cmd_Stop )
   END_RUNG
   RUNG wire#powerrail
      Contact( "UN".Alarm.sts_Category_3_Latched )
   END_RUNG wire#w1
   // the same network as SCL:
   "UN".PackML_Sts_Alarm.cmd_Stop := "UN".Alarm.sts_Category_2_Latched OR "UN".Alarm.sts_Category_3_Latched;
END_REGION

REGION Network 7: Hold Command - controlled by Category Alarm 7
   RUNG wire#powerrail
      Contact( "UN".Alarm.sts_Category_7_NotLatched )
      Coil( "UN".PackML_Sts_Alarm.cmd_Hold )
   END_RUNG
   // the same network as SCL:
   "UN".PackML_Sts_Alarm.cmd_Hold := "UN".Alarm.sts_Category_7_NotLatched;
END_REGION

REGION Network 8: UnHold Command - controlled by Category Alarm 7
   RUNG wire#powerrail
      Contact( "PackML".Sts.State.Held )
      I_Contact( "UN".Alarm.sts_Category_7_NotLatched )
      Coil( "UN".PackML_Sts_Alarm.cmd_UnHold )
   END_RUNG
   // the same network as SCL:
   "UN".PackML_Sts_Alarm.cmd_UnHold := "PackML".Sts.State.Held AND NOT "UN".Alarm.sts_Category_7_NotLatched;
END_REGION

REGION Network 9: Suspend Command - controlled by Category Alarm 8 or 9
   RUNG wire#powerrail
      Contact( "UN".Alarm.sts_Category_8_NotLatched )
      wire#w1
      Coil( "UN".PackML_Sts_Alarm.cmd_Suspend )
   END_RUNG
   RUNG wire#powerrail
      Contact( "UN".Alarm.sts_Category_9_NotLatched )
   END_RUNG wire#w1
   // the same network as SCL:
   "UN".PackML_Sts_Alarm.cmd_Suspend := "UN".Alarm.sts_Category_8_NotLatched OR "UN".Alarm.sts_Category_9_NotLatched;
END_REGION

REGION Network 10: UnSuspend Command - controlled by clearedCategory Alarm 8 or 9
   RUNG wire#powerrail
      Contact( "PackML".Sts.State.Suspended )
      I_Contact( "UN".Alarm.sts_Category_8_NotLatched )
      I_Contact( "UN".Alarm.sts_Category_9_NotLatched )
      Coil( "UN".PackML_Sts_Alarm.cmd_UnSuspend )
   END_RUNG
   // the same network as SCL:
   "UN".PackML_Sts_Alarm.cmd_UnSuspend := "PackML".Sts.State.Suspended AND NOT "UN".Alarm.sts_Category_8_NotLatched AND NOT "UN".Alarm.sts_Category_9_NotLatched;
END_REGION

REGION Network 11: Clearing SC Command - controlled by clearedCategory Alarm 0 or 1
   RUNG wire#powerrail
      Contact( "PackML".Sts.State.Clearing )
      I_Contact( "UN".Alarm.sts_Category_0_Latched )
      I_Contact( "UN".Alarm.sts_Category_1_Latched )
      Coil( "UN".PackML_Sts_Alarm.sts_Clearing_SC )
   END_RUNG
   // the same network as SCL:
   "UN".PackML_Sts_Alarm.sts_Clearing_SC := "PackML".Sts.State.Clearing AND NOT "UN".Alarm.sts_Category_0_Latched AND NOT "UN".Alarm.sts_Category_1_Latched;
END_REGION

REGION Network 12: Resetting S Command - controlled by clearedCategory Alarm 0-4
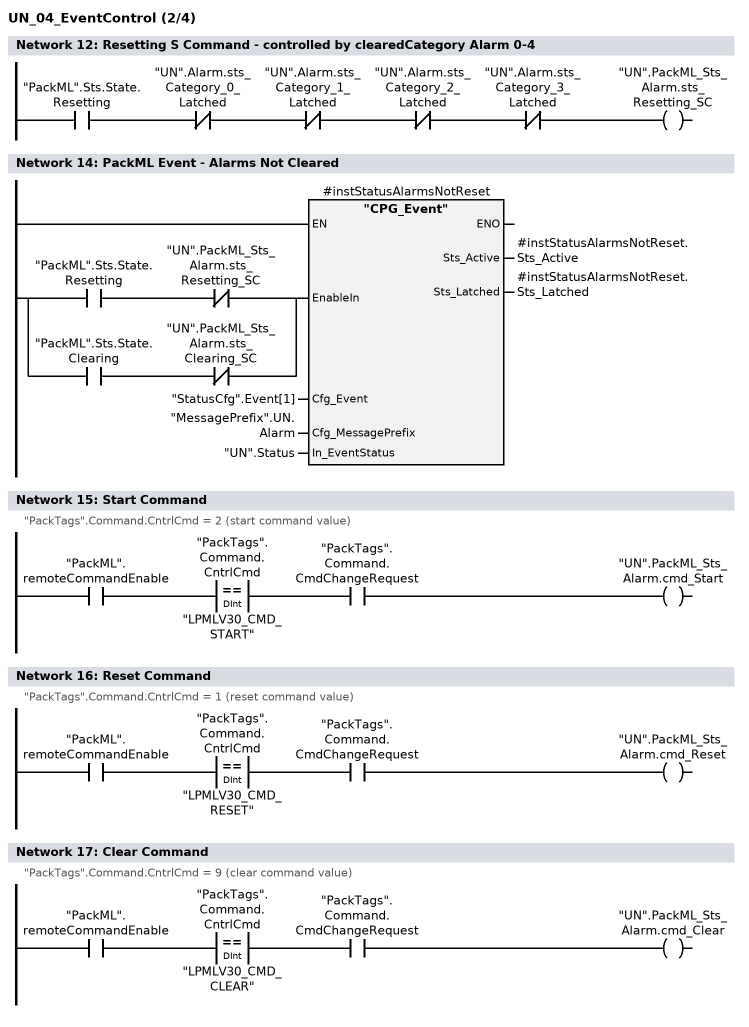
   RUNG wire#powerrail
      Contact( "PackML".Sts.State.Resetting )
      I_Contact( "UN".Alarm.sts_Category_0_Latched )
      I_Contact( "UN".Alarm.sts_Category_1_Latched )
      I_Contact( "UN".Alarm.sts_Category_2_Latched )
      I_Contact( "UN".Alarm.sts_Category_3_Latched )
      Coil( "UN".PackML_Sts_Alarm.sts_Resetting_SC )
   END_RUNG
   // the same network as SCL:
   "UN".PackML_Sts_Alarm.sts_Resetting_SC := "PackML".Sts.State.Resetting AND NOT "UN".Alarm.sts_Category_0_Latched AND NOT "UN".Alarm.sts_Category_1_Latched AND NOT "UN".Alarm.sts_Category_2_Latched AND NOT "UN".Alarm.sts_Category_3_Latched;
END_REGION

REGION Network 13: PackML Event -
END_REGION

